C09142=1180.504,309.494,-71.507,-176.660,7.868,148.547
C09143=1180.508,309.245,-71.477,-176.662,7.865,148.546
C09144=1180.512,308.997,-71.446,-176.664,7.862,148.546
C09145=1180.517,308.749,-71.415,-176.667,7.859,148.546
C09146=1180.521,308.501,-71.384,-176.669,7.855,148.546
C09147=1180.525,308.253,-71.354,-176.672,7.853,148.546
C09148=1180.529,308.005,-71.323,-176.674,7.850,148.546
C09149=1180.534,307.757,-71.292,-176.677,7.847,148.546
C09150=1180.537,307.509,-71.262,-176.679,7.844,148.546
C09151=1180.542,307.261,-71.231,-176.682,7.841,148.546
C09152=1180.546,307.013,-71.200,-176.685,7.838,148.546
C09153=1180.550,306.765,-71.170,-176.687,7.835,148.546
C09154=1180.555,306.516,-71.140,-176.690,7.832,148.546
C09155=1180.559,306.268,-71.109,-176.692,7.829,148.546
C09156=1180.563,306.020,-71.079,-176.695,7.826,148.546
C09157=1180.568,305.772,-71.048,-176.697,7.823,148.546
C09158=1180.572,305.525,-71.018,-176.700,7.820,148.546
C09159=1180.576,305.276,-70.987,-176.702,7.817,148.546
C09160=1180.580,305.027,-70.956,-176.705,7.814,148.546
C09161=1180.584,304.780,-70.926,-176.707,7.811,148.546
C09162=1180.589,304.532,-70.896,-176.710,7.808,148.546
C09163=1180.593,304.284,-70.865,-176.713,7.805,148.546
C09164=1180.597,304.035,-70.835,-176.716,7.802,148.546
C09165=1180.601,303.787,-70.805,-176.717,7.799,148.546
C09166=1180.606,303.539,-70.774,-176.720,7.796,148.546
C09167=1180.610,303.292,-70.744,-176.723,7.793,148.546
C09168=1180.614,303.043,-70.714,-176.725,7.790,148.546
C09169=1180.618,302.795,-70.684,-176.728,7.787,148.546
C09170=1180.622,302.547,-70.653,-176.730,7.784,148.546
C09171=1180.627,302.299,-70.623,-176.733,7.781,148.546
C09172=1180.631,302.051,-70.592,-176.736,7.778,148.546
C09173=1180.635,301.802,-70.563,-176.738,7.776,148.545
C09174=1180.640,301.554,-70.532,-176.740,7.773,148.545
C09175=1180.644,301.307,-70.502,-176.743,7.770,148.545
C09176=1180.649,301.058,-70.472,-176.746,7.767,148.545
C09177=1180.652,300.810,-70.441,-176.748,7.764,148.546
C09178=1180.657,300.561,-70.411,-176.751,7.760,148.545
C09179=1180.661,300.314,-70.381,-176.753,7.757,148.545
C09180=1180.666,300.065,-70.351,-176.756,7.755,148.545
C09181=1180.670,299.817,-70.321,-176.758,7.752,148.545
C09182=1180.674,299.569,-70.291,-176.761,7.749,148.545
C09183=1180.678,299.321,-70.261,-176.763,7.746,148.545
C09184=1180.683,299.073,-70.231,-176.766,7.743,148.545
C09185=1180.686,298.825,-70.201,-176.769,7.740,148.545
C09186=1180.691,298.576,-70.171,-176.771,7.737,148.545
C09187=1180.695,298.328,-70.140,-176.774,7.735,148.545
C09188=1180.700,298.080,-70.110,-176.776,7.731,148.545
C09189=1180.703,297.832,-70.080,-176.779,7.728,148.545
C09190=1180.708,297.584,-70.051,-176.781,7.726,148.545
C09191=1180.713,297.335,-70.021,-176.784,7.723,148.545
C09192=1180.716,297.088,-69.991,-176.787,7.720,148.545
C09193=1180.721,296.839,-69.961,-176.789,7.717,148.545
C09194=1180.725,296.591,-69.932,-176.791,7.714,148.545
C09195=1180.729,296.343,-69.901,-176.794,7.711,148.545
C09196=1180.734,296.095,-69.871,-176.797,7.708,148.545
C09197=1180.738,295.846,-69.842,-176.799,7.705,148.545
C09198=1180.742,295.599,-69.812,-176.802,7.702,148.545
C09199=1180.747,295.350,-69.782,-176.805,7.699,148.545
C09200=1180.751,295.102,-69.752,-176.807,7.697,148.545
C09201=1180.755,294.854,-69.722,-176.809,7.694,148.545
C09202=1180.759,294.606,-69.693,-176.812,7.691,148.545
C09203=1180.764,294.358,-69.663,-176.815,7.688,148.545
C09204=1180.768,294.109,-69.633,-176.817,7.685,148.545
C09205=1180.772,293.861,-69.604,-176.820,7.682,148.545
C09206=1180.776,293.613,-69.574,-176.822,7.680,148.545
C09207=1180.780,293.365,-69.544,-176.825,7.677,148.545
C09208=1180.785,293.116,-69.514,-176.827,7.673,148.545
C09209=1180.789,292.868,-69.485,-176.830,7.670,148.545
C09210=1180.793,292.620,-69.455,-176.833,7.667,148.545
C09211=1180.798,292.372,-69.426,-176.835,7.665,148.545
C09212=1180.801,292.124,-69.396,-176.838,7.662,148.545
C09213=1180.806,291.876,-69.366,-176.840,7.659,148.545
C09214=1180.810,291.627,-69.337,-176.843,7.656,148.545
C09215=1180.815,291.379,-69.307,-176.846,7.653,148.545
C09216=1180.819,291.131,-69.277,-176.848,7.650,148.545
C09217=1180.823,290.882,-69.248,-176.850,7.648,148.545
C09218=1180.827,290.634,-69.218,-176.853,7.645,148.545
C09219=1180.832,290.387,-69.189,-176.856,7.642,148.545
C09220=1180.836,290.138,-69.160,-176.858,7.639,148.545
C09221=1180.840,289.890,-69.130,-176.861,7.636,148.546
C09222=1180.845,289.642,-69.101,-176.863,7.634,148.546
C09223=1180.849,289.393,-69.071,-176.866,7.631,148.546
C09224=1180.853,289.145,-69.042,-176.869,7.628,148.546
C09225=1180.857,288.897,-69.012,-176.871,7.625,148.546
C09226=1180.863,288.622,-68.980,-176.874,7.622,148.546
C09227=1180.867,288.348,-68.947,-176.877,7.619,148.546
C09228=1180.872,288.072,-68.915,-176.880,7.616,148.546
C09229=1180.876,287.799,-68.883,-176.883,7.612,148.546
C09230=1180.881,287.550,-68.854,-176.885,7.610,148.546
C09231=1180.885,287.302,-68.824,-176.888,7.607,148.546
C09232=1180.889,287.053,-68.795,-176.890,7.603,148.546
C09233=1180.894,286.806,-68.766,-176.893,7.600,148.546
C09234=1180.898,286.557,-68.736,-176.896,7.597,148.546
C09235=1180.902,286.309,-68.707,-176.898,7.595,148.546
C09236=1180.907,286.060,-68.678,-176.900,7.592,148.546
C09237=1180.911,285.812,-68.649,-176.903,7.589,148.546
C09238=1180.915,285.564,-68.619,-176.906,7.586,148.546
C09239=1180.920,285.316,-68.590,-176.909,7.583,148.546
C09240=1180.924,285.067,-68.561,-176.911,7.581,148.546
C09241=1180.928,284.819,-68.532,-176.913,7.578,148.546
C09242=1180.933,284.571,-68.503,-176.916,7.575,148.546
C09243=1180.937,284.322,-68.473,-176.919,7.572,148.546
C09244=1180.941,284.075,-68.445,-176.921,7.570,148.546
C09245=1180.945,283.826,-68.416,-176.924,7.567,148.546
C09246=1180.949,283.578,-68.386,-176.927,7.564,148.546
C09247=1180.954,283.329,-68.358,-176.929,7.561,148.546
C09248=1180.959,283.082,-68.329,-176.932,7.558,148.546
C09249=1180.963,282.833,-68.299,-176.934,7.556,148.546
C09250=1180.967,282.584,-68.270,-176.937,7.553,148.546
C09251=1180.971,282.337,-68.241,-176.940,7.550,148.546
C09252=1180.976,282.088,-68.213,-176.942,7.547,148.547
C09253=1180.980,281.840,-68.184,-176.945,7.545,148.547
C09254=1180.984,281.592,-68.154,-176.947,7.542,148.547
C09255=1180.989,281.343,-68.125,-176.950,7.539,148.547
C09256=1180.993,281.096,-68.097,-176.953,7.536,148.547
C09257=1180.997,280.847,-68.068,-176.955,7.534,148.547
C09258=1181.001,280.598,-68.039,-176.958,7.531,148.547
C09259=1181.006,280.350,-68.010,-176.960,7.528,148.547
C09260=1181.010,280.102,-67.982,-176.963,7.525,148.547
C09261=1181.014,279.853,-67.953,-176.965,7.522,148.547
C09262=1181.019,279.605,-67.923,-176.968,7.520,148.547
C09263=1181.024,279.357,-67.895,-176.971,7.517,148.547
C09264=1181.027,279.109,-67.866,-176.973,7.514,148.547
C09265=1181.032,278.860,-67.837,-176.976,7.511,148.547
C09266=1181.037,278.612,-67.809,-176.978,7.508,148.547
C09267=1181.040,278.364,-67.780,-176.981,7.505,148.547
C09268=1181.045,278.115,-67.751,-176.984,7.502,148.547
C09269=1181.049,277.868,-67.722,-176.986,7.500,148.547
C09270=1181.053,277.619,-67.694,-176.989,7.497,148.547
C09271=1181.058,277.370,-67.665,-176.991,7.494,148.547
C09272=1181.063,277.123,-67.636,-176.994,7.491,148.548
C09273=1181.066,276.874,-67.608,-176.996,7.489,148.548
C09274=1181.071,276.625,-67.579,-176.999,7.486,148.548
C09275=1181.075,276.377,-67.552,-177.002,7.483,148.548
C09276=1181.079,276.129,-67.522,-177.004,7.481,148.548
C09277=1181.084,275.880,-67.494,-177.007,7.478,148.548
C09278=1181.088,275.632,-67.466,-177.009,7.475,148.548
C09279=1181.092,275.384,-67.436,-177.012,7.472,148.548
C09280=1181.097,275.136,-67.409,-177.014,7.470,148.548
C09281=1181.101,274.887,-67.380,-177.017,7.467,148.548
C09282=1181.105,274.639,-67.352,-177.020,7.464,148.548
C09283=1181.110,274.390,-67.323,-177.022,7.462,148.548
C09284=1181.114,274.142,-67.294,-177.025,7.459,148.548
C09285=1181.119,273.894,-67.266,-177.027,7.456,148.548
C09286=1181.123,273.645,-67.237,-177.030,7.453,148.548
C09287=1181.127,273.397,-67.210,-177.032,7.451,148.548
C09288=1181.132,273.149,-67.181,-177.035,7.448,148.549
C09289=1181.136,272.900,-67.153,-177.038,7.445,148.549
C09290=1181.141,272.652,-67.124,-177.040,7.443,148.549
C09291=1181.144,272.404,-67.095,-177.043,7.440,148.549
C09292=1181.149,272.156,-67.067,-177.046,7.437,148.549
C09293=1181.153,271.907,-67.039,-177.049,7.434,148.549
C09294=1181.157,271.659,-67.011,-177.051,7.432,148.549
C09295=1181.162,271.410,-66.982,-177.053,7.429,148.549
C09296=1181.166,271.162,-66.955,-177.056,7.426,148.549
C09297=1181.171,270.914,-66.926,-177.058,7.424,148.549
C09298=1181.175,270.666,-66.898,-177.061,7.421,148.549
C09299=1181.179,270.417,-66.869,-177.064,7.418,148.549
C09300=1181.184,270.169,-66.842,-177.066,7.416,148.549
C09301=1181.188,269.920,-66.813,-177.069,7.413,148.550
C09302=1181.193,269.672,-66.785,-177.072,7.410,148.550
C09303=1181.196,269.424,-66.757,-177.074,7.408,148.550
C09304=1181.201,269.175,-66.729,-177.077,7.405,148.550
C09305=1181.205,268.927,-66.700,-177.080,7.402,148.550
C09306=1181.210,268.678,-66.673,-177.082,7.399,148.550
C09307=1181.214,268.429,-66.645,-177.084,7.397,148.550
C09308=1181.219,268.182,-66.617,-177.087,7.394,148.550
C09309=1181.222,267.933,-66.589,-177.090,7.391,148.550
C09310=1181.228,267.685,-66.560,-177.093,7.389,148.550
C09311=1181.231,267.436,-66.532,-177.095,7.386,148.550
C09312=1181.236,267.188,-66.504,-177.098,7.383,148.550
C09313=1181.241,266.940,-66.477,-177.100,7.381,148.550
C09314=1181.245,266.691,-66.449,-177.103,7.378,148.551
C09315=1181.249,266.443,-66.421,-177.106,7.375,148.551
C09316=1181.254,266.194,-66.392,-177.108,7.373,148.551
C09317=1181.258,265.946,-66.365,-177.111,7.370,148.551
C09318=1181.262,265.697,-66.337,-177.114,7.367,148.551
C09319=1181.266,265.449,-66.309,-177.116,7.365,148.551
C09320=1181.271,265.201,-66.281,-177.119,7.362,148.551
C09321=1181.276,264.952,-66.253,-177.121,7.359,148.551
C09322=1181.280,264.704,-66.226,-177.124,7.357,148.551
C09323=1181.284,264.456,-66.198,-177.126,7.354,148.551
C09324=1181.289,264.207,-66.170,-177.129,7.352,148.552
C09325=1181.293,263.959,-66.142,-177.132,7.349,148.552
C09326=1181.297,263.710,-66.114,-177.134,7.346,148.552
C09327=1181.302,263.462,-66.087,-177.137,7.344,148.552
C09328=1181.306,263.214,-66.059,-177.139,7.341,148.552
C09329=1181.310,262.965,-66.031,-177.142,7.338,148.552
C09330=1181.315,262.693,-66.001,-177.145,7.335,148.552
C09331=1181.320,262.419,-65.970,-177.148,7.332,148.552
C09332=1181.325,262.147,-65.940,-177.151,7.329,148.552
C09333=1181.330,261.873,-65.909,-177.154,7.327,148.553
C09334=1181.334,261.625,-65.882,-177.156,7.324,148.553
C09335=1181.338,261.376,-65.854,-177.159,7.321,148.553
C09336=1181.343,261.128,-65.827,-177.161,7.318,148.553
C09337=1181.347,260.880,-65.799,-177.164,7.316,148.553
C09338=1181.351,260.631,-65.771,-177.167,7.314,148.553
C09339=1181.356,260.383,-65.744,-177.169,7.311,148.553
C09340=1181.361,260.134,-65.716,-177.172,7.308,148.553
C09341=1181.365,259.886,-65.688,-177.174,7.306,148.553
C09342=1181.369,259.637,-65.661,-177.177,7.303,148.553
C09343=1181.374,259.389,-65.633,-177.180,7.301,148.554
C09344=1181.378,259.141,-65.606,-177.183,7.298,148.554
C09345=1181.382,258.891,-65.578,-177.185,7.296,148.554
C09346=1181.387,258.643,-65.551,-177.188,7.293,148.554
C09347=1181.391,258.395,-65.524,-177.190,7.290,148.554
C09348=1181.396,258.147,-65.496,-177.193,7.288,148.554
C09349=1181.400,257.898,-65.468,-177.196,7.285,148.554
C09350=1181.405,257.649,-65.441,-177.198,7.283,148.554
C09351=1181.409,257.402,-65.414,-177.201,7.280,148.554
C09352=1181.414,257.153,-65.387,-177.203,7.278,148.555
C09353=1181.418,256.904,-65.359,-177.206,7.275,148.555
C09354=1181.422,256.655,-65.332,-177.209,7.272,148.555
C09355=1181.427,256.407,-65.304,-177.211,7.270,148.555
C09356=1181.431,256.159,-65.277,-177.214,7.267,148.555
C09357=1181.435,255.910,-65.250,-177.216,7.265,148.555
C09358=1181.440,255.662,-65.222,-177.219,7.262,148.555
C09359=1181.444,255.414,-65.196,-177.222,7.259,148.555
C09360=1181.448,255.165,-65.168,-177.224,7.257,148.555
C09361=1181.453,254.917,-65.141,-177.227,7.254,148.556
C09362=1181.457,254.668,-65.114,-177.229,7.252,148.556
C09363=1181.461,254.420,-65.086,-177.232,7.249,148.556
C09364=1181.466,254.171,-65.059,-177.235,7.246,148.556
C09365=1181.471,253.923,-65.032,-177.237,7.244,148.556
C09366=1181.475,253.674,-65.005,-177.240,7.241,148.556
C09367=1181.480,253.426,-64.978,-177.242,7.239,148.556
C09368=1181.483,253.177,-64.951,-177.245,7.236,148.557
C09369=1181.488,252.928,-64.924,-177.248,7.234,148.557
C09370=1181.492,252.680,-64.896,-177.250,7.231,148.557
C09371=1181.497,252.432,-64.869,-177.253,7.228,148.557
C09372=1181.502,252.183,-64.842,-177.256,7.227,148.557
C09373=1181.506,251.935,-64.815,-177.258,7.224,148.557
C09374=1181.510,251.687,-64.789,-177.261,7.221,148.557
C09375=1181.514,251.438,-64.761,-177.263,7.218,148.557
C09376=1181.519,251.189,-64.734,-177.266,7.217,148.558
C09377=1181.524,250.941,-64.707,-177.269,7.214,148.558
C09378=1181.527,250.692,-64.681,-177.271,7.211,148.558
C09379=1181.532,250.444,-64.654,-177.274,7.209,148.558
C09380=1181.537,250.195,-64.626,-177.277,7.206,148.558
C09381=1181.541,249.947,-64.599,-177.279,7.204,148.558
C09382=1181.545,249.699,-64.573,-177.282,7.201,148.559
C09383=1181.550,249.450,-64.546,-177.284,7.199,148.559
C09384=1181.555,249.202,-64.519,-177.287,7.196,148.559
C09385=1181.559,248.952,-64.492,-177.290,7.194,148.559
C09386=1181.563,248.704,-64.466,-177.293,7.191,148.559
C09387=1181.568,248.455,-64.439,-177.295,7.189,148.559
C09388=1181.572,248.207,-64.412,-177.297,7.186,148.559
C09389=1181.576,247.959,-64.385,-177.300,7.184,148.560
C09390=1181.581,247.710,-64.358,-177.303,7.181,148.560
C09391=1181.585,247.462,-64.331,-177.306,7.178,148.560
C09392=1181.590,247.213,-64.305,-177.308,7.176,148.560
C09393=1181.594,246.964,-64.278,-177.311,7.173,148.560
C09394=1181.599,246.716,-64.251,-177.313,7.171,148.560
C09395=1181.603,246.468,-64.225,-177.316,7.169,148.560
C09396=1181.608,246.219,-64.198,-177.318,7.167,148.561
C09397=1181.612,245.970,-64.172,-177.322,7.164,148.561
C09398=1181.616,245.722,-64.145,-177.324,7.162,148.561
C09399=1181.621,245.473,-64.118,-177.327,7.159,148.561
C09400=1181.625,245.225,-64.091,-177.329,7.157,148.561
C09401=1181.630,244.976,-64.065,-177.332,7.154,148.561
C09402=1181.634,244.728,-64.038,-177.334,7.152,148.561
C09403=1181.639,244.479,-64.011,-177.337,7.149,148.562
C09404=1181.644,244.230,-63.985,-177.340,7.147,148.562
C09405=1181.647,243.982,-63.959,-177.342,7.144,148.562
C09406=1181.652,243.734,-63.931,-177.345,7.142,148.562
C09407=1181.656,243.485,-63.906,-177.348,7.139,148.562
C09408=1181.661,243.236,-63.879,-177.350,7.137,148.563
C09409=1181.665,242.988,-63.852,-177.353,7.134,148.563
C09410=1181.670,242.739,-63.826,-177.355,7.132,148.563
C09411=1181.674,242.491,-63.799,-177.358,7.130,148.563
C09412=1181.679,242.242,-63.773,-177.361,7.128,148.563
C09413=1181.683,241.993,-63.747,-177.363,7.125,148.563
C09414=1181.688,241.744,-63.720,-177.366,7.123,148.564
C09415=1181.692,241.496,-63.694,-177.369,7.120,148.564
C09416=1181.697,241.248,-63.667,-177.371,7.118,148.564
C09417=1181.701,241.000,-63.641,-177.374,7.115,148.564
C09418=1181.705,240.751,-63.615,-177.376,7.113,148.564
C09419=1181.710,240.502,-63.588,-177.379,7.110,148.564
C09420=1181.714,240.254,-63.562,-177.382,7.108,148.565
C09421=1181.719,240.005,-63.536,-177.385,7.105,148.565
C09422=1181.723,239.756,-63.510,-177.387,7.103,148.565
C09423=1181.728,239.508,-63.483,-177.390,7.100,148.565
C09424=1181.732,239.259,-63.457,-177.392,7.098,148.565
C09425=1181.736,239.011,-63.431,-177.395,7.095,148.565
C09426=1181.741,238.762,-63.405,-177.398,7.094,148.566
C09427=1181.745,238.514,-63.378,-177.401,7.091,148.566
C09428=1181.750,238.265,-63.352,-177.403,7.089,148.566
C09429=1181.754,238.016,-63.326,-177.405,7.087,148.566
C09430=1181.758,237.768,-63.300,-177.408,7.084,148.566
C09431=1181.763,237.519,-63.273,-177.411,7.082,148.567
C09432=1181.768,237.270,-63.248,-177.414,7.079,148.567
C09433=1181.772,237.023,-63.221,-177.416,7.077,148.567
C09434=1181.778,236.750,-63.193,-177.419,7.074,148.567
C09435=1181.782,236.479,-63.164,-177.422,7.072,148.567
C09436=1181.787,236.207,-63.136,-177.425,7.069,148.567
C09437=1181.791,235.936,-63.107,-177.428,7.067,148.568
C09438=1181.797,235.687,-63.081,-177.431,7.064,148.568
C09439=1181.801,235.439,-63.056,-177.433,7.062,148.568
C09440=1181.805,235.190,-63.030,-177.436,7.059,148.568
C09441=1181.809,234.942,-63.003,-177.438,7.057,148.568
C09442=1181.814,234.693,-62.977,-177.441,7.054,148.569
C09443=1181.819,234.444,-62.952,-177.444,7.052,148.569
C09444=1181.823,234.196,-62.926,-177.446,7.050,148.569
C09445=1181.827,233.947,-62.900,-177.449,7.048,148.569
C09446=1181.832,233.698,-62.874,-177.451,7.045,148.569
C09447=1181.836,233.450,-62.847,-177.454,7.043,148.570
C09448=1181.841,233.201,-62.822,-177.457,7.041,148.570
C09449=1181.845,232.953,-62.796,-177.460,7.038,148.570
C09450=1181.849,232.704,-62.770,-177.462,7.036,148.570
C09451=1181.854,232.455,-62.744,-177.465,7.033,148.570
C09452=1181.859,232.207,-62.719,-177.467,7.031,148.571
C09453=1181.863,231.958,-62.693,-177.470,7.029,148.571
C09454=1181.868,231.709,-62.667,-177.473,7.026,148.571
C09455=1181.872,231.461,-62.642,-177.475,7.025,148.571
C09456=1181.877,231.212,-62.616,-177.478,7.022,148.571
C09457=1181.881,230.963,-62.590,-177.481,7.020,148.572
C09458=1181.886,230.714,-62.564,-177.483,7.018,148.572
C09459=1181.891,230.466,-62.539,-177.486,7.015,148.572
C09460=1181.895,230.217,-62.513,-177.488,7.013,148.572
C09461=1181.899,229.968,-62.487,-177.492,7.010,148.573
C09462=1181.904,229.720,-62.462,-177.494,7.008,148.573
C09463=1181.908,229.472,-62.436,-177.496,7.006,148.573
C09464=1181.912,229.223,-62.410,-177.499,7.003,148.573
C09465=1181.917,228.974,-62.384,-177.502,7.001,148.573
C09466=1181.921,228.726,-62.359,-177.505,6.999,148.573
C09467=1181.926,228.477,-62.333,-177.507,6.997,148.574
C09468=1181.930,228.228,-62.308,-177.509,6.995,148.574
C09469=1181.935,227.980,-62.282,-177.513,6.992,148.574
C09470=1181.939,227.731,-62.256,-177.515,6.990,148.574
C09471=1181.944,227.483,-62.232,-177.518,6.987,148.575
C09472=1181.948,227.234,-62.206,-177.521,6.985,148.575
C09473=1181.952,226.985,-62.180,-177.523,6.983,148.575
C09474=1181.957,226.737,-62.155,-177.526,6.981,148.575
C09475=1181.962,226.488,-62.129,-177.528,6.978,148.575
C09476=1181.966,226.239,-62.103,-177.532,6.976,148.576
C09477=1181.971,225.991,-62.079,-177.534,6.974,148.576
C09478=1181.975,225.742,-62.053,-177.536,6.972,148.576
C09479=1181.979,225.493,-62.027,-177.539,6.969,148.576
C09480=1181.984,225.245,-62.002,-177.542,6.967,148.577
C09481=1181.989,224.995,-61.977,-177.544,6.965,148.577
C09482=1181.994,224.747,-61.951,-177.547,6.962,148.577
C09483=1181.998,224.498,-61.926,-177.550,6.960,148.577
C09484=1182.003,224.250,-61.900,-177.553,6.958,148.577
C09485=1182.007,224.001,-61.875,-177.555,6.956,148.578
C09486=1182.011,223.752,-61.849,-177.557,6.954,148.578
C09487=1182.016,223.504,-61.824,-177.561,6.951,148.578
C09488=1182.021,223.255,-61.799,-177.563,6.949,148.578
C09489=1182.025,223.007,-61.774,-177.565,6.947,148.579
C09490=1182.029,222.757,-61.749,-177.569,6.944,148.579
C09491=1182.034,222.509,-61.724,-177.571,6.942,148.579
C09492=1182.038,222.260,-61.698,-177.574,6.940,148.579
C09493=1182.043,222.011,-61.673,-177.576,6.937,148.579
C09494=1182.048,221.763,-61.648,-177.579,6.936,148.580
C09495=1182.052,221.514,-61.623,-177.582,6.933,148.580
C09496=1182.056,221.266,-61.598,-177.584,6.931,148.580
C09497=1182.061,221.017,-61.572,-177.587,6.929,148.580
C09498=1182.066,220.768,-61.547,-177.590,6.926,148.581
C09499=1182.070,220.519,-61.522,-177.592,6.924,148.581
C09500=1182.074,220.271,-61.498,-177.595,6.922,148.581
C09501=1182.079,220.022,-61.472,-177.598,6.919,148.581
C09502=1182.084,219.773,-61.447,-177.600,6.918,148.582
C09503=1182.088,219.525,-61.421,-177.603,6.916,148.582
C09504=1182.093,219.276,-61.397,-177.606,6.913,148.582
C09505=1182.097,219.027,-61.372,-177.608,6.911,148.582
C09506=1182.102,218.779,-61.347,-177.611,6.909,148.582
C09507=1182.106,218.529,-61.322,-177.614,6.906,148.583
C09508=1182.110,218.282,-61.297,-177.617,6.905,148.583
C09509=1182.115,218.032,-61.272,-177.619,6.902,148.583
C09510=1182.120,217.784,-61.247,-177.622,6.900,148.584
C09511=1182.124,217.535,-61.222,-177.625,6.898,148.584
C09512=1182.129,217.286,-61.198,-177.627,6.896,148.584
C09513=1182.133,217.038,-61.172,-177.630,6.893,148.584
C09514=1182.138,216.789,-61.147,-177.632,6.891,148.584
C09515=1182.142,216.540,-61.123,-177.635,6.889,148.585
C09516=1182.147,216.291,-61.097,-177.638,6.887,148.585
C09517=1182.152,216.043,-61.073,-177.640,6.884,148.585
C09518=1182.155,215.794,-61.048,-177.643,6.883,148.586
C09519=1182.160,215.545,-61.023,-177.646,6.880,148.586
C09520=1182.165,215.297,-60.998,-177.648,6.878,148.586
C09521=1182.169,215.048,-60.974,-177.651,6.876,148.586
C09522=1182.174,214.799,-60.949,-177.654,6.874,148.587
C09523=1182.178,214.550,-60.924,-177.656,6.871,148.587
C09524=1182.183,214.302,-60.899,-177.659,6.870,148.587
C09525=1182.188,214.053,-60.875,-177.662,6.868,148.587
C09526=1182.192,213.804,-60.850,-177.664,6.865,148.587
C09527=1182.197,213.555,-60.825,-177.667,6.863,148.588
C09528=1182.200,213.307,-60.800,-177.670,6.861,148.588
C09529=1182.206,213.058,-60.776,-177.673,6.858,148.588
C09530=1182.210,212.809,-60.751,-177.675,6.856,148.589
C09531=1182.215,212.560,-60.726,-177.678,6.855,148.589
C09532=1182.219,212.312,-60.702,-177.680,6.852,148.589
C09533=1182.224,212.063,-60.678,-177.683,6.850,148.589
C09534=1182.229,211.813,-60.653,-177.686,6.848,148.590
C09535=1182.233,211.566,-60.628,-177.688,6.846,148.590
C09536=1182.238,211.317,-60.603,-177.691,6.843,148.590
C09537=1182.242,211.068,-60.579,-177.694,6.841,148.590
C09538=1182.247,210.798,-60.552,-177.697,6.840,148.591
C09539=1182.252,210.527,-60.526,-177.699,6.837,148.591
C09540=1182.257,210.256,-60.499,-177.703,6.834,148.591
C09541=1182.262,209.986,-60.472,-177.705,6.832,148.592
C09542=1182.266,209.737,-60.448,-177.708,6.831,148.592
C09543=1182.271,209.489,-60.424,-177.711,6.828,148.592
C09544=1182.275,209.240,-60.399,-177.713,6.826,148.592
C09545=1182.280,208.991,-60.375,-177.716,6.824,148.593
C09546=1182.285,208.742,-60.350,-177.719,6.822,148.593
C09547=1182.289,208.493,-60.326,-177.721,6.819,148.593
C09548=1182.294,208.245,-60.301,-177.724,6.817,148.593
C09549=1182.298,207.996,-60.277,-177.727,6.816,148.594
C09550=1182.302,207.748,-60.253,-177.729,6.813,148.594
C09551=1182.307,207.498,-60.228,-177.732,6.811,148.594
C09552=1182.312,207.249,-60.205,-177.735,6.809,148.595
C09553=1182.317,207.001,-60.180,-177.737,6.807,148.595
C09554=1182.321,206.752,-60.156,-177.740,6.804,148.595
C09555=1182.325,206.503,-60.132,-177.743,6.802,148.595
C09556=1182.330,206.254,-60.107,-177.746,6.801,148.596
C09557=1182.335,206.006,-60.083,-177.748,6.799,148.596
C09558=1182.339,205.758,-60.059,-177.751,6.796,148.596
C09559=1182.344,205.508,-60.035,-177.754,6.794,148.596
C09560=1182.348,205.259,-60.010,-177.756,6.792,148.597
C09561=1182.353,205.011,-59.986,-177.758,6.790,148.597
C09562=1182.358,204.762,-59.962,-177.762,6.788,148.597
C09563=1182.362,204.513,-59.938,-177.764,6.786,148.598
C09564=1182.367,204.265,-59.914,-177.767,6.784,148.598
C09565=1182.371,204.015,-59.890,-177.769,6.782,148.598
C09566=1182.376,203.767,-59.865,-177.772,6.780,148.598
C09567=1182.380,203.518,-59.842,-177.775,6.777,148.599
C09568=1182.385,203.269,-59.818,-177.778,6.776,148.599
C09569=1182.389,203.021,-59.794,-177.780,6.774,148.599
C09570=1182.394,202.771,-59.768,-177.783,6.772,148.599
C09571=1182.398,202.522,-59.745,-177.786,6.769,148.600
C09572=1182.403,202.274,-59.721,-177.788,6.767,148.600
C09573=1182.407,202.026,-59.697,-177.791,6.765,148.600
C09574=1182.413,201.776,-59.673,-177.793,6.763,148.601
C09575=1182.417,201.528,-59.649,-177.796,6.762,148.601
C09576=1182.422,201.279,-59.626,-177.799,6.759,148.601
C09577=1182.426,201.030,-59.601,-177.801,6.757,148.601
C09578=1182.430,200.781,-59.577,-177.804,6.755,148.602
C09579=1182.435,200.532,-59.554,-177.807,6.753,148.602
C09580=1182.440,200.283,-59.529,-177.810,6.751,148.602
C09581=1182.444,200.034,-59.506,-177.812,6.748,148.603
C09582=1182.449,199.786,-59.482,-177.815,6.747,148.603
C09583=1182.454,199.537,-59.458,-177.818,6.745,148.603
C09584=1182.458,199.289,-59.434,-177.820,6.743,148.604
C09585=1182.463,199.040,-59.411,-177.823,6.740,148.604
C09586=1182.466,198.790,-59.386,-177.826,6.738,148.604
C09587=1182.472,198.541,-59.362,-177.828,6.737,148.604
C09588=1182.476,198.293,-59.338,-177.831,6.735,148.605
C09589=1182.481,198.044,-59.315,-177.834,6.733,148.605
C09590=1182.485,197.795,-59.291,-177.836,6.731,148.605
C09591=1182.490,197.546,-59.268,-177.839,6.728,148.606
C09592=1182.494,197.298,-59.243,-177.842,6.726,148.606
C09593=1182.499,197.049,-59.220,-177.844,6.725,148.606
C09594=1182.504,196.800,-59.197,-177.847,6.723,148.607
C09595=1182.508,196.551,-59.173,-177.849,6.721,148.607
C09596=1182.513,196.302,-59.149,-177.852,6.718,148.607
C09597=1182.517,196.054,-59.125,-177.855,6.716,148.607
C09598=1182.522,195.805,-59.102,-177.858,6.715,148.608
C09599=1182.527,195.556,-59.079,-177.860,6.712,148.608
C09600=1182.531,195.307,-59.054,-177.863,6.711,148.608
C09601=1182.536,195.058,-59.031,-177.865,6.709,148.609
C09602=1182.541,194.809,-59.008,-177.869,6.706,148.609
C09603=1182.545,194.561,-58.984,-177.871,6.704,148.609
C09604=1182.550,194.312,-58.960,-177.874,6.703,148.610
C09605=1182.554,194.063,-58.937,-177.876,6.700,148.610
C09606=1182.559,193.814,-58.914,-177.879,6.699,148.610
C09607=1182.563,193.565,-58.890,-177.881,6.697,148.610
C09608=1182.568,193.316,-58.866,-177.885,6.694,148.611
C09609=1182.573,193.067,-58.843,-177.887,6.692,148.611
C09610=1182.578,192.818,-58.819,-177.889,6.690,148.611
C09611=1182.582,192.570,-58.795,-177.892,6.689,148.612
C09612=1182.587,192.321,-58.772,-177.895,6.687,148.612
C09613=1182.591,192.072,-58.749,-177.897,6.685,148.612
C09614=1182.596,191.823,-58.725,-177.901,6.682,148.613
C09615=1182.600,191.574,-58.703,-177.903,6.681,148.613
C09616=1182.605,191.325,-58.679,-177.906,6.678,148.613
C09617=1182.609,191.077,-58.655,-177.908,6.677,148.613
C09618=1182.614,190.828,-58.632,-177.911,6.675,148.614
C09619=1182.619,190.579,-58.608,-177.914,6.673,148.614
C09620=1182.623,190.330,-58.585,-177.916,6.671,148.614
C09621=1182.628,190.080,-58.562,-177.919,6.669,148.615
C09622=1182.632,189.832,-58.539,-177.922,6.667,148.615
C09623=1182.637,189.583,-58.516,-177.924,6.665,148.615
C09624=1182.642,189.334,-58.493,-177.927,6.663,148.616
C09625=1182.647,189.085,-58.469,-177.930,6.661,148.616
C09626=1182.651,188.836,-58.446,-177.932,6.659,148.616
C09627=1182.656,188.587,-58.422,-177.935,6.658,148.617
C09628=1182.660,188.339,-58.400,-177.938,6.656,148.617
C09629=1182.665,188.090,-58.376,-177.940,6.653,148.617
C09630=1182.669,187.841,-58.353,-177.943,6.651,148.617
C09631=1182.675,187.592,-58.330,-177.946,6.649,148.618
C09632=1182.679,187.343,-58.307,-177.948,6.648,148.618
C09633=1182.683,187.094,-58.284,-177.951,6.646,148.619
C09634=1182.688,186.845,-58.261,-177.954,6.644,148.619
C09635=1182.693,186.596,-58.237,-177.956,6.642,148.619
C09636=1182.697,186.348,-58.214,-177.959,6.640,148.619
C09637=1182.701,186.099,-58.191,-177.961,6.638,148.620
C09638=1182.707,185.850,-58.168,-177.965,6.636,148.620
C09639=1182.711,185.601,-58.145,-177.967,6.634,148.620
C09640=1182.715,185.353,-58.122,-177.970,6.632,148.621
C09641=1182.720,185.104,-58.099,-177.973,6.630,148.621
C09642=1182.725,184.834,-58.074,-177.975,6.628,148.622
C09643=1182.730,184.564,-58.049,-177.979,6.626,148.622
C09644=1182.735,184.295,-58.024,-177.981,6.624,148.622
C09645=1182.740,184.025,-58.000,-177.984,6.622,148.623
C09646=1182.745,183.776,-57.976,-177.987,6.621,148.623
C09647=1182.749,183.527,-57.953,-177.989,6.619,148.623
C09648=1182.754,183.278,-57.931,-177.992,6.616,148.624
C09649=1182.759,183.029,-57.908,-177.995,6.614,148.624
C09650=1182.763,182.780,-57.884,-177.997,6.612,148.624
C09651=1182.767,182.532,-57.862,-178.000,6.610,148.624
C09652=1182.772,182.282,-57.839,-178.003,6.609,148.625
C09653=1182.777,182.034,-57.817,-178.005,6.607,148.625
C09654=1182.782,181.785,-57.793,-178.008,6.605,148.626
C09655=1182.787,181.535,-57.771,-178.011,6.603,148.626
C09656=1182.791,181.287,-57.748,-178.013,6.602,148.626
C09657=1182.796,181.038,-57.725,-178.016,6.600,148.627
C09658=1182.800,180.789,-57.702,-178.019,6.598,148.627
C09659=1182.805,180.540,-57.680,-178.021,6.596,148.627
C09660=1182.809,180.291,-57.657,-178.024,6.593,148.627
C09661=1182.814,180.043,-57.634,-178.027,6.591,148.628
C09662=1182.818,179.793,-57.612,-178.029,6.590,148.628
C09663=1182.823,179.544,-57.588,-178.032,6.588,148.629
C09664=1182.828,179.296,-57.567,-178.035,6.586,148.629
C09665=1182.833,179.047,-57.543,-178.037,6.584,148.629
C09666=1182.837,178.798,-57.521,-178.040,6.583,148.630
C09667=1182.842,178.548,-57.498,-178.043,6.581,148.630
C09668=1182.846,178.300,-57.475,-178.046,6.579,148.630
C09669=1182.851,178.051,-57.453,-178.048,6.577,148.631
C09670=1182.855,177.802,-57.430,-178.051,6.575,148.631
C09671=1182.861,177.553,-57.408,-178.054,6.574,148.631
C09672=1182.865,177.304,-57.385,-178.056,6.572,148.632
C09673=1182.870,177.055,-57.362,-178.059,6.570,148.632
C09674=1182.874,176.807,-57.340,-178.061,6.568,148.632
C09675=1182.879,176.557,-57.317,-178.064,6.566,148.633
C09676=1182.883,176.308,-57.295,-178.066,6.564,148.633
C09677=1182.888,176.060,-57.273,-178.069,6.563,148.633
C09678=1182.893,175.811,-57.250,-178.072,6.561,148.634
C09679=1182.897,175.561,-57.228,-178.074,6.559,148.634
C09680=1182.902,175.313,-57.205,-178.078,6.556,148.634
C09681=1182.907,175.064,-57.182,-178.080,6.555,148.635
C09682=1182.911,174.814,-57.160,-178.083,6.553,148.635
C09683=1182.916,174.566,-57.137,-178.086,6.551,148.635
C09684=1182.921,174.317,-57.115,-178.088,6.549,148.636
C09685=1182.926,174.068,-57.092,-178.091,6.548,148.636
C09686=1182.930,173.819,-57.070,-178.094,6.546,148.637
C09687=1182.934,173.570,-57.048,-178.096,6.544,148.637
C09688=1182.940,173.321,-57.025,-178.099,6.542,148.637
C09689=1182.944,173.072,-57.003,-178.102,6.540,148.638
C09690=1182.949,172.823,-56.982,-178.104,6.539,148.638
C09691=1182.954,172.574,-56.959,-178.107,6.537,148.638
C09692=1182.958,172.325,-56.936,-178.110,6.535,148.639
C09693=1182.963,172.076,-56.914,-178.113,6.533,148.639
C09694=1182.967,171.827,-56.892,-178.115,6.532,148.639
C09695=1182.972,171.579,-56.869,-178.118,6.530,148.640
C09696=1182.977,171.329,-56.847,-178.121,6.528,148.640
C09697=1182.981,171.081,-56.826,-178.123,6.526,148.641
C09698=1182.986,170.831,-56.803,-178.125,6.524,148.641
C09699=1182.991,170.583,-56.781,-178.128,6.522,148.641
C09700=1182.995,170.334,-56.759,-178.131,6.521,148.641
C09701=1183.000,170.084,-56.737,-178.133,6.519,148.642
C09702=1183.005,169.835,-56.714,-178.136,6.517,148.642
C09703=1183.009,169.586,-56.692,-178.139,6.515,148.643
C09704=1183.014,169.337,-56.671,-178.141,6.513,148.643
C09705=1183.018,169.089,-56.648,-178.144,6.512,148.643
C09706=1183.023,168.840,-56.626,-178.147,6.510,148.644
C09707=1183.028,168.590,-56.603,-178.150,6.508,148.644
C09708=1183.033,168.342,-56.582,-178.152,6.506,148.644
C09709=1183.037,168.092,-56.560,-178.155,6.505,148.645
C09710=1183.042,167.844,-56.538,-178.158,6.503,148.645
C09711=1183.046,167.594,-56.516,-178.160,6.501,148.646
C09712=1183.052,167.345,-56.494,-178.163,6.499,148.646
C09713=1183.056,167.096,-56.472,-178.166,6.497,148.646
C09714=1183.061,166.847,-56.450,-178.168,6.496,148.647
C09715=1183.065,166.598,-56.428,-178.171,6.494,148.647
C09716=1183.070,166.349,-56.406,-178.174,6.492,148.647
C09717=1183.075,166.100,-56.384,-178.176,6.490,148.648
C09718=1183.079,165.852,-56.362,-178.179,6.489,148.648
C09719=1183.084,165.603,-56.340,-178.182,6.487,148.648
C09720=1183.089,165.353,-56.318,-178.184,6.486,148.649
C09721=1183.094,165.104,-56.297,-178.187,6.484,148.649
C09722=1183.098,164.855,-56.274,-178.190,6.483,148.650
C09723=1183.103,164.606,-56.253,-178.192,6.481,148.650
C09724=1183.108,164.357,-56.231,-178.195,6.479,148.651
C09725=1183.112,164.108,-56.209,-178.198,6.477,148.651
C09726=1183.117,163.859,-56.187,-178.200,6.476,148.651
C09727=1183.122,163.610,-56.165,-178.203,6.474,148.652
C09728=1183.126,163.362,-56.144,-178.206,6.472,148.652
C09729=1183.131,163.113,-56.122,-178.208,6.470,148.652
C09730=1183.136,162.864,-56.100,-178.211,6.468,148.653
C09731=1183.140,162.615,-56.078,-178.214,6.467,148.653
C09732=1183.145,162.365,-56.057,-178.216,6.465,148.653
C09733=1183.150,162.117,-56.035,-178.219,6.463,148.654
C09734=1183.154,161.867,-56.013,-178.222,6.461,148.654
C09735=1183.159,161.619,-55.991,-178.224,6.460,148.655
C09736=1183.163,161.369,-55.969,-178.227,6.458,148.655
C09737=1183.168,161.121,-55.948,-178.230,6.456,148.655
C09738=1183.173,160.871,-55.927,-178.233,6.454,148.656
C09739=1183.178,160.622,-55.905,-178.235,6.453,148.656
C09740=1183.182,160.373,-55.883,-178.237,6.452,148.656
C09741=1183.187,160.125,-55.861,-178.240,6.450,148.657
C09742=1183.192,159.875,-55.840,-178.243,6.448,148.657
C09743=1183.197,159.626,-55.818,-178.245,6.446,148.658
C09744=1183.202,159.378,-55.797,-178.248,6.445,148.658
C09745=1183.206,159.128,-55.775,-178.251,6.443,148.659
C09746=1183.211,158.859,-55.752,-178.254,6.441,148.659
C09747=1183.216,158.590,-55.729,-178.257,6.440,148.659
C09748=1183.221,158.321,-55.706,-178.260,6.437,148.660
C09749=1183.227,158.053,-55.682,-178.263,6.435,148.660
C09750=1183.230,157.803,-55.661,-178.266,6.434,148.661
C09751=1183.235,157.554,-55.640,-178.268,6.433,148.661
C09752=1183.240,157.306,-55.618,-178.270,6.431,148.661
C09753=1183.245,157.056,-55.597,-178.273,6.429,148.662
C09754=1183.250,156.807,-55.575,-178.276,6.428,148.662
C09755=1183.255,156.558,-55.554,-178.279,6.426,148.663
C09756=1183.259,156.310,-55.533,-178.281,6.424,148.663
C09757=1183.263,156.060,-55.511,-178.284,6.422,148.663
C09758=1183.268,155.811,-55.490,-178.287,6.420,148.664
C09759=1183.273,155.562,-55.468,-178.289,6.419,148.664
C09760=1183.278,155.312,-55.447,-178.292,6.417,148.664
C09761=1183.283,155.064,-55.425,-178.294,6.416,148.665
C09762=1183.287,154.815,-55.405,-178.297,6.414,148.665
C09763=1183.292,154.566,-55.383,-178.300,6.413,148.666
C09764=1183.297,154.316,-55.362,-178.303,6.411,148.666
C09765=1183.301,154.068,-55.340,-178.305,6.409,148.667
C09766=1183.306,153.819,-55.320,-178.308,6.407,148.667
C09767=1183.311,153.570,-55.298,-178.311,6.406,148.667
C09768=1183.316,153.321,-55.277,-178.313,6.404,148.668
C09769=1183.320,153.071,-55.255,-178.316,6.402,148.668
C09770=1183.325,152.822,-55.235,-178.318,6.401,148.668
C09771=1183.330,152.574,-55.213,-178.321,6.399,148.669
C09772=1183.335,152.325,-55.192,-178.324,6.398,148.669
C09773=1183.340,152.075,-55.171,-178.327,6.396,148.670
C09774=1183.343,151.826,-55.150,-178.329,6.395,148.670
C09775=1183.349,151.577,-55.129,-178.332,6.393,148.671
C09776=1183.353,151.328,-55.107,-178.335,6.391,148.671
C09777=1183.358,151.079,-55.087,-178.337,6.389,148.671
C09778=1183.363,150.830,-55.066,-178.340,6.388,148.672
C09779=1183.367,150.581,-55.044,-178.342,6.387,148.672
C09780=1183.372,150.332,-55.023,-178.345,6.385,148.672
C09781=1183.377,150.083,-55.002,-178.348,6.383,148.673
C09782=1183.382,149.834,-54.981,-178.351,6.382,148.673
C09783=1183.386,149.585,-54.960,-178.353,6.380,148.674
C09784=1183.391,149.336,-54.939,-178.356,6.378,148.674
C09785=1183.396,149.086,-54.918,-178.358,6.377,148.675
C09786=1183.400,148.837,-54.897,-178.361,6.375,148.675
C09787=1183.405,148.588,-54.876,-178.364,6.374,148.675
C09788=1183.410,148.339,-54.855,-178.366,6.372,148.676
C09789=1183.415,148.090,-54.834,-178.370,6.370,148.676
C09790=1183.420,147.841,-54.813,-178.372,6.369,148.677
C09791=1183.424,147.592,-54.792,-178.375,6.367,148.677
C09792=1183.429,147.343,-54.771,-178.377,6.366,148.677
C09793=1183.433,147.093,-54.751,-178.380,6.364,148.678
C09794=1183.438,146.844,-54.730,-178.382,6.362,148.678
C09795=1183.443,146.596,-54.709,-178.385,6.361,148.679
C09796=1183.448,146.347,-54.688,-178.388,6.359,148.679
C09797=1183.452,146.098,-54.667,-178.391,6.357,148.680
C09798=1183.457,145.848,-54.646,-178.393,6.357,148.680
C09799=1183.462,145.599,-54.626,-178.396,6.355,148.680
C09800=1183.467,145.350,-54.605,-178.398,6.353,148.681
C09801=1183.471,145.101,-54.585,-178.401,6.351,148.681
C09802=1183.476,144.853,-54.563,-178.404,6.350,148.682
C09803=1183.481,144.604,-54.543,-178.407,6.348,148.682
C09804=1183.486,144.354,-54.522,-178.409,6.347,148.683
C09805=1183.490,144.105,-54.501,-178.412,6.345,148.683
C09806=1183.495,143.855,-54.480,-178.414,6.344,148.683
C09807=1183.499,143.607,-54.460,-178.417,6.342,148.684
C09808=1183.504,143.357,-54.439,-178.420,6.340,148.684
C09809=1183.509,143.108,-54.418,-178.422,6.340,148.685
C09810=1183.514,142.859,-54.397,-178.425,6.338,148.685
C09811=1183.519,142.610,-54.377,-178.428,6.336,148.685
C09812=1183.524,142.361,-54.356,-178.431,6.334,148.686
C09813=1183.528,142.112,-54.336,-178.433,6.332,148.686
C09814=1183.533,141.863,-54.315,-178.435,6.332,148.687
C09815=1183.538,141.614,-54.294,-178.439,6.330,148.687
C09816=1183.542,141.365,-54.274,-178.441,6.328,148.688
C09817=1183.547,141.116,-54.253,-178.444,6.327,148.688
C09818=1183.552,140.867,-54.232,-178.447,6.325,148.688
C09819=1183.556,140.618,-54.212,-178.449,6.324,148.689
C09820=1183.562,140.368,-54.192,-178.451,6.322,148.689
C09821=1183.566,140.119,-54.171,-178.455,6.321,148.690
C09822=1183.571,139.870,-54.151,-178.457,6.319,148.690
C09823=1183.576,139.621,-54.130,-178.460,6.317,148.691
C09824=1183.580,139.372,-54.110,-178.462,6.316,148.691
C09825=1183.585,139.123,-54.089,-178.465,6.315,148.691
C09826=1183.590,138.873,-54.068,-178.468,6.313,148.692
C09827=1183.594,138.624,-54.048,-178.471,6.311,148.692
C09828=1183.599,138.375,-54.028,-178.473,6.310,148.693
C09829=1183.604,138.126,-54.007,-178.475,6.309,148.693
C09830=1183.609,137.877,-53.987,-178.478,6.307,148.694
C09831=1183.614,137.628,-53.967,-178.481,6.306,148.694
C09832=1183.618,137.380,-53.947,-178.484,6.304,148.695
C09833=1183.624,137.130,-53.926,-178.486,6.303,148.695
C09834=1183.628,136.881,-53.906,-178.489,6.301,148.695
C09835=1183.632,136.632,-53.886,-178.492,6.299,148.696
C09836=1183.638,136.382,-53.865,-178.495,6.298,148.696
C09837=1183.642,136.133,-53.845,-178.497,6.297,148.697
C09838=1183.647,135.884,-53.825,-178.500,6.295,148.697
C09839=1183.651,135.635,-53.804,-178.502,6.293,148.698
C09840=1183.656,135.385,-53.785,-178.505,6.292,148.698
C09841=1183.661,135.136,-53.764,-178.508,6.290,148.698
C09842=1183.666,134.888,-53.744,-178.510,6.289,148.699
C09843=1183.671,134.638,-53.724,-178.513,6.288,148.699
C09844=1183.675,134.389,-53.704,-178.516,6.286,148.700
C09845=1183.680,134.140,-53.683,-178.519,6.284,148.700
C09846=1183.685,133.891,-53.663,-178.521,6.284,148.701
C09847=1183.690,133.642,-53.643,-178.524,6.282,148.701
C09848=1183.694,133.393,-53.622,-178.526,6.280,148.701
C09849=1183.700,133.144,-53.603,-178.529,6.278,148.702
C09850=1183.704,132.875,-53.580,-178.532,6.277,148.702
C09851=1183.709,132.606,-53.559,-178.534,6.276,148.703
C09852=1183.715,132.337,-53.537,-178.537,6.275,148.704
C09853=1183.719,132.069,-53.516,-178.540,6.273,148.704
C09854=1183.725,131.820,-53.496,-178.543,6.271,148.704
C09855=1183.729,131.571,-53.476,-178.546,6.270,148.705
C09856=1183.735,131.321,-53.456,-178.549,6.268,148.705
C09857=1183.739,131.072,-53.435,-178.551,6.267,148.706
C09858=1183.744,130.823,-53.416,-178.554,6.265,148.706
C09859=1183.748,130.574,-53.395,-178.557,6.264,148.707
C09860=1183.754,130.325,-53.376,-178.559,6.263,148.707
C09861=1183.758,130.076,-53.356,-178.562,6.261,148.707
C09862=1183.763,129.827,-53.336,-178.564,6.259,148.708
C09863=1183.767,129.578,-53.316,-178.567,6.258,148.709
C09864=1183.773,129.329,-53.296,-178.570,6.257,148.709
C09865=1183.777,129.080,-53.276,-178.572,6.255,148.709
C09866=1183.782,128.830,-53.256,-178.575,6.254,148.710
C09867=1183.787,128.581,-53.237,-178.578,6.252,148.710
C09868=1183.791,128.332,-53.216,-178.580,6.251,148.711
C09869=1183.796,128.083,-53.197,-178.583,6.249,148.711
C09870=1183.801,127.834,-53.177,-178.586,6.248,148.712
C09871=1183.806,127.584,-53.157,-178.588,6.247,148.712
C09872=1183.810,127.335,-53.137,-178.591,6.245,148.713
C09873=1183.815,127.087,-53.117,-178.594,6.244,148.713
C09874=1183.820,126.837,-53.098,-178.596,6.243,148.713
C09875=1183.825,126.587,-53.078,-178.599,6.241,148.714
C09876=1183.829,126.338,-53.058,-178.602,6.240,148.714
C09877=1183.835,126.090,-53.038,-178.604,6.238,148.715
C09878=1183.839,125.840,-53.019,-178.606,6.237,148.715
C09879=1183.844,125.591,-52.998,-178.610,6.235,148.716
C09880=1183.849,125.342,-52.979,-178.612,6.234,148.716
C09881=1183.854,125.093,-52.959,-178.614,6.233,148.717
C09882=1183.859,124.843,-52.940,-178.618,6.231,148.717
C09883=1183.863,124.594,-52.919,-178.620,6.230,148.718
C09884=1183.868,124.345,-52.900,-178.623,6.229,148.718
C09885=1183.873,124.096,-52.880,-178.625,6.227,148.718
C09886=1183.878,123.846,-52.861,-178.628,6.226,148.719
C09887=1183.882,123.598,-52.841,-178.631,6.225,148.719
C09888=1183.887,123.349,-52.822,-178.633,6.223,148.720
C09889=1183.892,123.099,-52.802,-178.636,6.222,148.720
C09890=1183.897,122.850,-52.783,-178.639,6.220,148.721
C09891=1183.902,122.601,-52.763,-178.641,6.219,148.721
C09892=1183.906,122.351,-52.743,-178.644,6.217,148.722
C09893=1183.911,122.103,-52.723,-178.647,6.216,148.722
C09894=1183.915,121.854,-52.704,-178.649,6.215,148.723
C09895=1183.920,121.604,-52.685,-178.652,6.213,148.723
C09896=1183.926,121.355,-52.665,-178.655,6.212,148.724
C09897=1183.930,121.106,-52.646,-178.657,6.211,148.724
C09898=1183.935,120.856,-52.626,-178.660,6.209,148.724
C09899=1183.940,120.607,-52.607,-178.663,6.208,148.725
C09900=1183.944,120.358,-52.588,-178.665,6.207,148.726
C09901=1183.950,120.109,-52.568,-178.668,6.205,148.726
C09902=1183.955,119.859,-52.549,-178.671,6.203,148.726
C09903=1183.959,119.610,-52.528,-178.673,6.203,148.727
C09904=1183.964,119.362,-52.510,-178.676,6.201,148.727
C09905=1183.968,119.112,-52.490,-178.678,6.200,148.728
C09906=1183.973,118.863,-52.470,-178.681,6.199,148.728
C09907=1183.978,118.614,-52.451,-178.684,6.197,148.729
C09908=1183.983,118.364,-52.431,-178.686,6.196,148.729
C09909=1183.988,118.116,-52.413,-178.689,6.194,148.730
C09910=1183.992,117.866,-52.393,-178.692,6.193,148.730
C09911=1183.998,117.617,-52.374,-178.694,6.192,148.731
C09912=1184.002,117.367,-52.355,-178.697,6.190,148.731
C09913=1184.007,117.118,-52.336,-178.700,6.189,148.732
C09914=1184.012,116.869,-52.317,-178.702,6.188,148.732
C09915=1184.017,116.619,-52.297,-178.705,6.186,148.733
C09916=1184.022,116.371,-52.278,-178.708,6.185,148.733
C09917=1184.026,116.121,-52.259,-178.710,6.184,148.734
C09918=1184.032,115.872,-52.239,-178.713,6.182,148.734
C09919=1184.036,115.623,-52.220,-178.715,6.181,148.735
C09920=1184.041,115.374,-52.201,-178.718,6.180,148.735
C09921=1184.046,115.125,-52.181,-178.721,6.178,148.736
C09922=1184.051,114.876,-52.163,-178.724,6.177,148.736
C09923=1184.055,114.626,-52.144,-178.726,6.176,148.736
C09924=1184.061,114.377,-52.124,-178.729,6.174,148.737
C09925=1184.065,114.128,-52.105,-178.732,6.173,148.737
C09926=1184.070,113.879,-52.086,-178.734,6.172,148.738
C09927=1184.074,113.630,-52.067,-178.737,6.171,148.738
C09928=1184.080,113.380,-52.048,-178.740,6.169,148.739
C09929=1184.084,113.131,-52.029,-178.742,6.168,148.739
C09930=1184.089,112.882,-52.010,-178.745,6.167,148.740
C09931=1184.094,112.633,-51.990,-178.748,6.165,148.740
C09932=1184.099,112.383,-51.972,-178.750,6.164,148.741
C09933=1184.103,112.134,-51.953,-178.753,6.163,148.741
C09934=1184.109,111.885,-51.933,-178.756,6.161,148.742
C09935=1184.113,111.636,-51.914,-178.758,6.160,148.742
C09936=1184.118,111.386,-51.896,-178.761,6.159,148.743
C09937=1184.122,111.137,-51.877,-178.763,6.158,148.743
C09938=1184.128,110.888,-51.857,-178.766,6.156,148.744
C09939=1184.132,110.638,-51.839,-178.769,6.155,148.744
C09940=1184.137,110.389,-51.820,-178.771,6.154,148.745
C09941=1184.141,110.140,-51.801,-178.774,6.153,148.745
C09942=1184.147,109.891,-51.782,-178.776,6.152,148.746
C09943=1184.152,109.642,-51.763,-178.779,6.150,148.746
C09944=1184.156,109.392,-51.744,-178.782,6.148,148.747
C09945=1184.161,109.143,-51.726,-178.784,6.148,148.747
C09946=1184.166,108.894,-51.706,-178.787,6.146,148.748
C09947=1184.171,108.645,-51.688,-178.790,6.145,148.748
C09948=1184.176,108.395,-51.669,-178.792,6.144,148.749
C09949=1184.180,108.146,-51.650,-178.795,6.142,148.749
C09950=1184.186,107.897,-51.631,-178.798,6.141,148.750
C09951=1184.190,107.648,-51.612,-178.800,6.139,148.750
C09952=1184.196,107.398,-51.594,-178.803,6.139,148.751
C09953=1184.200,107.150,-51.575,-178.806,6.137,148.751
C09954=1184.206,106.880,-51.555,-178.809,6.136,148.752
C09955=1184.210,106.613,-51.534,-178.811,6.135,148.752
C09956=1184.216,106.344,-51.514,-178.814,6.134,148.753
C09957=1184.220,106.076,-51.494,-178.817,6.132,148.753
C09958=1184.226,105.826,-51.475,-178.820,6.131,148.754
C09959=1184.231,105.578,-51.457,-178.822,6.129,148.754
C09960=1184.236,105.328,-51.438,-178.825,6.128,148.755
C09961=1184.241,105.078,-51.420,-178.828,6.127,148.755
C09962=1184.245,104.829,-51.401,-178.830,6.125,148.756
C09963=1184.250,104.580,-51.382,-178.833,6.125,148.756
C09964=1184.255,104.331,-51.363,-178.836,6.123,148.757
C09965=1184.259,104.081,-51.345,-178.838,6.122,148.757
C09966=1184.264,103.832,-51.326,-178.841,6.121,148.758
C09967=1184.269,103.583,-51.308,-178.843,6.120,148.758
C09968=1184.274,103.333,-51.289,-178.846,6.118,148.759
C09969=1184.279,103.084,-51.270,-178.849,6.117,148.759
C09970=1184.284,102.835,-51.252,-178.851,6.116,148.760
C09971=1184.289,102.586,-51.234,-178.854,6.115,148.760
C09972=1184.294,102.337,-51.215,-178.857,6.114,148.761
C09973=1184.298,102.087,-51.197,-178.859,6.112,148.761
C09974=1184.303,101.839,-51.178,-178.862,6.111,148.762
C09975=1184.308,101.589,-51.159,-178.865,6.110,148.762
C09976=1184.313,101.339,-51.141,-178.867,6.109,148.763
C09977=1184.318,101.090,-51.123,-178.870,6.107,148.763
C09978=1184.322,100.841,-51.104,-178.873,6.107,148.764
C09979=1184.328,100.592,-51.085,-178.875,6.105,148.764
C09980=1184.333,100.342,-51.067,-178.878,6.103,148.765
C09981=1184.337,100.094,-51.049,-178.881,6.103,148.765
C09982=1184.341,99.844,-51.030,-178.883,6.101,148.766
C09983=1184.347,99.594,-51.012,-178.886,6.100,148.766
C09984=1184.352,99.345,-50.994,-178.889,6.099,148.767
C09985=1184.357,99.097,-50.975,-178.891,6.098,148.767
C09986=1184.361,98.847,-50.957,-178.894,6.096,148.768
C09987=1184.366,98.598,-50.939,-178.896,6.096,148.768
C09988=1184.371,98.348,-50.920,-178.899,6.094,148.769
C09989=1184.376,98.099,-50.902,-178.901,6.093,148.769
C09990=1184.381,97.849,-50.884,-178.905,6.092,148.770
C09991=1184.385,97.601,-50.865,-178.907,6.091,148.770
C09992=1184.390,97.351,-50.847,-178.909,6.089,148.771
C09993=1184.395,97.102,-50.829,-178.912,6.089,148.771
C09994=1184.401,96.853,-50.811,-178.915,6.087,148.772
C09995=1184.405,96.603,-50.792,-178.917,6.086,148.773
C09996=1184.410,96.354,-50.774,-178.920,6.085,148.773
//INST
///DATE 2021/06/15 17:24
///ATTR SC,RW,RJ
////FRAME ROBOT
///GROUP1 RB1
NOP
MOVL C00000 V=800.0 PL=0
MOVL C00001 V=800.0 PL=0
MOVL C00002 V=800.0 PL=0
MOVL C00003 V=800.0 PL=0
MOVL C00004 V=800.0 PL=0
MOVL C00005 V=800.0 PL=0
MOVL C00006 V=800.0 PL=0
MOVL C00007 V=800.0 PL=0
MOVL C00008 V=800.0 PL=0
MOVL C00009 V=800.0 PL=0
MOVL C00010 V=800.0 PL=0
MOVL C00011 V=800.0 PL=0
MOVL C00012 V=800.0 PL=0
MOVL C00013 V=800.0 PL=0
MOVL C00014 V=800.0 PL=0
MOVL C00015 V=800.0 PL=0
MOVL C00016 V=800.0 PL=0
MOVL C00017 V=800.0 PL=0
MOVL C00018 V=800.0 PL=0
MOVL C00019 V=800.0 PL=0
MOVL C00020 V=800.0 PL=0
MOVL C00021 V=800.0 PL=0
MOVL C00022 V=800.0 PL=0
MOVL C00023 V=800.0 PL=0
MOVL C00024 V=800.0 PL=0
MOVL C00025 V=800.0 PL=0
MOVL C00026 V=800.0 PL=0
MOVL C00027 V=800.0 PL=0
MOVL C00028 V=800.0 PL=0
MOVL C00029 V=800.0 PL=0
MOVL C00030 V=800.0 PL=0
MOVL C00031 V=800.0 PL=0
MOVL C00032 V=800.0 PL=0
MOVL C00033 V=800.0 PL=0
MOVL C00034 V=800.0 PL=0
MOVL C00035 V=800.0 PL=0
MOVL C00036 V=800.0 PL=0
MOVL C00037 V=800.0 PL=0
MOVL C00038 V=800.0 PL=0
MOVL C00039 V=800.0 PL=0
MOVL C00040 V=800.0 PL=0
MOVL C00041 V=800.0 PL=0
MOVL C00042 V=800.0 PL=0
MOVL C00043 V=800.0 PL=0
MOVL C00044 V=800.0 PL=0
MOVL C00045 V=800.0 PL=0
MOVL C00046 V=800.0 PL=0
MOVL C00047 V=800.0 PL=0
MOVL C00048 V=800.0 PL=0
MOVL C00049 V=800.0 PL=0
MOVL C00050 V=800.0 PL=0
MOVL C00051 V=800.0 PL=0
MOVL C00052 V=800.0 PL=0
MOVL C00053 V=800.0 PL=0
MOVL C00054 V=800.0 PL=0
MOVL C00055 V=800.0 PL=0
MOVL C00056 V=800.0 PL=0
MOVL C00057 V=800.0 PL=0
MOVL C00058 V=800.0 PL=0
MOVL C00059 V=800.0 PL=0
MOVL C00060 V=800.0 PL=0
MOVL C00061 V=800.0 PL=0
MOVL C00062 V=800.0 PL=0
MOVL C00063 V=800.0 PL=0
MOVL C00064 V=800.0 PL=0
MOVL C00065 V=800.0 PL=0
MOVL C00066 V=800.0 PL=0
MOVL C00067 V=800.0 PL=0
MOVL C00068 V=800.0 PL=0
MOVL C00069 V=800.0 PL=0
MOVL C00070 V=800.0 PL=0
MOVL C00071 V=800.0 PL=0
MOVL C00072 V=800.0 PL=0
MOVL C00073 V=800.0 PL=0
MOVL C00074 V=800.0 PL=0
MOVL C00075 V=800.0 PL=0
MOVL C00076 V=800.0 PL=0
MOVL C00077 V=800.0 PL=0
MOVL C00078 V=800.0 PL=0
MOVL C00079 V=800.0 PL=0
MOVL C00080 V=800.0 PL=0
MOVL C00081 V=800.0 PL=0
MOVL C00082 V=800.0 PL=0
MOVL C00083 V=800.0 PL=0
MOVL C00084 V=800.0 PL=0
MOVL C00085 V=800.0 PL=0
MOVL C00086 V=800.0 PL=0
MOVL C00087 V=800.0 PL=0
MOVL C00088 V=800.0 PL=0
MOVL C00089 V=800.0 PL=0
MOVL C00090 V=800.0 PL=0
MOVL C00091 V=800.0 PL=0
MOVL C00092 V=800.0 PL=0
MOVL C00093 V=800.0 PL=0
MOVL C00094 V=800.0 PL=0
MOVL C00095 V=800.0 PL=0
MOVL C00096 V=800.0 PL=0
MOVL C00097 V=800.0 PL=0
MOVL C00098 V=800.0 PL=0
MOVL C00099 V=800.0 PL=0
MOVL C00100 V=800.0 PL=0
MOVL C00101 V=800.0 PL=0
MOVL C00102 V=800.0 PL=0
MOVL C00103 V=800.0 PL=0
MOVL C00104 V=800.0 PL=0
MOVL C00105 V=800.0 PL=0
MOVL C00106 V=800.0 PL=0
MOVL C00107 V=800.0 PL=0
MOVL C00108 V=800.0 PL=0
MOVL C00109 V=800.0 PL=0
MOVL C00110 V=800.0 PL=0
MOVL C00111 V=800.0 PL=0
MOVL C00112 V=800.0 PL=0
MOVL C00113 V=800.0 PL=0
MOVL C00114 V=800.0 PL=0
MOVL C00115 V=800.0 PL=0
MOVL C00116 V=800.0 PL=0
MOVL C00117 V=800.0 PL=0
MOVL C00118 V=800.0 PL=0
MOVL C00119 V=800.0 PL=0
MOVL C00120 V=800.0 PL=0
MOVL C00121 V=800.0 PL=0
MOVL C00122 V=800.0 PL=0
MOVL C00123 V=800.0 PL=0
MOVL C00124 V=800.0 PL=0
MOVL C00125 V=800.0 PL=0
MOVL C00126 V=800.0 PL=0
MOVL C00127 V=800.0 PL=0
MOVL C00128 V=800.0 PL=0
MOVL C00129 V=800.0 PL=0
MOVL C00130 V=800.0 PL=0
MOVL C00131 V=800.0 PL=0
MOVL C00132 V=800.0 PL=0
MOVL C00133 V=800.0 PL=0
MOVL C00134 V=800.0 PL=0
MOVL C00135 V=800.0 PL=0
MOVL C00136 V=800.0 PL=0
MOVL C00137 V=800.0 PL=0
MOVL C00138 V=800.0 PL=0
MOVL C00139 V=800.0 PL=0
MOVL C00140 V=800.0 PL=0
MOVL C00141 V=800.0 PL=0
MOVL C00142 V=800.0 PL=0
MOVL C00143 V=800.0 PL=0
MOVL C00144 V=800.0 PL=0
MOVL C00145 V=800.0 PL=0
MOVL C00146 V=800.0 PL=0
MOVL C00147 V=800.0 PL=0
MOVL C00148 V=800.0 PL=0
MOVL C00149 V=800.0 PL=0
MOVL C00150 V=800.0 PL=0
MOVL C00151 V=800.0 PL=0
MOVL C00152 V=800.0 PL=0
MOVL C00153 V=800.0 PL=0
MOVL C00154 V=800.0 PL=0
MOVL C00155 V=800.0 PL=0
MOVL C00156 V=800.0 PL=0
MOVL C00157 V=800.0 PL=0
MOVL C00158 V=800.0 PL=0
MOVL C00159 V=800.0 PL=0
MOVL C00160 V=800.0 PL=0
MOVL C00161 V=800.0 PL=0
MOVL C00162 V=800.0 PL=0
MOVL C00163 V=800.0 PL=0
MOVL C00164 V=800.0 PL=0
MOVL C00165 V=800.0 PL=0
MOVL C00166 V=800.0 PL=0
MOVL C00167 V=800.0 PL=0
MOVL C00168 V=800.0 PL=0
MOVL C00169 V=800.0 PL=0
MOVL C00170 V=800.0 PL=0
MOVL C00171 V=800.0 PL=0
MOVL C00172 V=800.0 PL=0
MOVL C00173 V=800.0 PL=0
MOVL C00174 V=800.0 PL=0
MOVL C00175 V=800.0 PL=0
MOVL C00176 V=800.0 PL=0
MOVL C00177 V=800.0 PL=0
MOVL C00178 V=800.0 PL=0
MOVL C00179 V=800.0 PL=0
MOVL C00180 V=800.0 PL=0
MOVL C00181 V=800.0 PL=0
MOVL C00182 V=800.0 PL=0
MOVL C00183 V=800.0 PL=0
MOVL C00184 V=800.0 PL=0
MOVL C00185 V=800.0 PL=0
MOVL C00186 V=800.0 PL=0
MOVL C00187 V=800.0 PL=0
MOVL C00188 V=800.0 PL=0
MOVL C00189 V=800.0 PL=0
MOVL C00190 V=800.0 PL=0
MOVL C00191 V=800.0 PL=0
MOVL C00192 V=800.0 PL=0
MOVL C00193 V=800.0 PL=0
MOVL C00194 V=800.0 PL=0
MOVL C00195 V=800.0 PL=0
MOVL C00196 V=800.0 PL=0
MOVL C00197 V=800.0 PL=0
MOVL C00198 V=800.0 PL=0
MOVL C00199 V=800.0 PL=0
MOVL C00200 V=800.0 PL=0
MOVL C00201 V=800.0 PL=0
MOVL C00202 V=800.0 PL=0
MOVL C00203 V=800.0 PL=0
MOVL C00204 V=800.0 PL=0
MOVL C00205 V=800.0 PL=0
MOVL C00206 V=800.0 PL=0
MOVL C00207 V=800.0 PL=0
MOVL C00208 V=800.0 PL=0
MOVL C00209 V=800.0 PL=0
MOVL C00210 V=800.0 PL=0
MOVL C00211 V=800.0 PL=0
MOVL C00212 V=800.0 PL=0
MOVL C00213 V=800.0 PL=0
MOVL C00214 V=800.0 PL=0
MOVL C00215 V=800.0 PL=0
MOVL C00216 V=800.0 PL=0
MOVL C00217 V=800.0 PL=0
MOVL C00218 V=800.0 PL=0
MOVL C00219 V=800.0 PL=0
MOVL C00220 V=800.0 PL=0
MOVL C00221 V=800.0 PL=0
MOVL C00222 V=800.0 PL=0
MOVL C00223 V=800.0 PL=0
MOVL C00224 V=800.0 PL=0
MOVL C00225 V=800.0 PL=0
MOVL C00226 V=800.0 PL=0
MOVL C00227 V=800.0 PL=0
MOVL C00228 V=800.0 PL=0
MOVL C00229 V=800.0 PL=0
MOVL C00230 V=800.0 PL=0
MOVL C00231 V=800.0 PL=0
MOVL C00232 V=800.0 PL=0
MOVL C00233 V=800.0 PL=0
MOVL C00234 V=800.0 PL=0
MOVL C00235 V=800.0 PL=0
MOVL C00236 V=800.0 PL=0
MOVL C00237 V=800.0 PL=0
MOVL C00238 V=800.0 PL=0
MOVL C00239 V=800.0 PL=0
MOVL C00240 V=800.0 PL=0
MOVL C00241 V=800.0 PL=0
MOVL C00242 V=800.0 PL=0
MOVL C00243 V=800.0 PL=0
MOVL C00244 V=800.0 PL=0
MOVL C00245 V=800.0 PL=0
MOVL C00246 V=800.0 PL=0
MOVL C00247 V=800.0 PL=0
MOVL C00248 V=800.0 PL=0
MOVL C00249 V=800.0 PL=0
MOVL C00250 V=800.0 PL=0
MOVL C00251 V=800.0 PL=0
MOVL C00252 V=800.0 PL=0
MOVL C00253 V=800.0 PL=0
MOVL C00254 V=800.0 PL=0
MOVL C00255 V=800.0 PL=0
MOVL C00256 V=800.0 PL=0
MOVL C00257 V=800.0 PL=0
MOVL C00258 V=800.0 PL=0
MOVL C00259 V=800.0 PL=0
MOVL C00260 V=800.0 PL=0
MOVL C00261 V=800.0 PL=0
MOVL C00262 V=800.0 PL=0
MOVL C00263 V=800.0 PL=0
MOVL C00264 V=800.0 PL=0
MOVL C00265 V=800.0 PL=0
MOVL C00266 V=800.0 PL=0
MOVL C00267 V=800.0 PL=0
MOVL C00268 V=800.0 PL=0
MOVL C00269 V=800.0 PL=0
MOVL C00270 V=800.0 PL=0
MOVL C00271 V=800.0 PL=0
MOVL C00272 V=800.0 PL=0
MOVL C00273 V=800.0 PL=0
MOVL C00274 V=800.0 PL=0
MOVL C00275 V=800.0 PL=0
MOVL C00276 V=800.0 PL=0
MOVL C00277 V=800.0 PL=0
MOVL C00278 V=800.0 PL=0
MOVL C00279 V=800.0 PL=0
MOVL C00280 V=800.0 PL=0
MOVL C00281 V=800.0 PL=0
MOVL C00282 V=800.0 PL=0
MOVL C00283 V=800.0 PL=0
MOVL C00284 V=800.0 PL=0
MOVL C00285 V=800.0 PL=0
MOVL C00286 V=800.0 PL=0
MOVL C00287 V=800.0 PL=0
MOVL C00288 V=800.0 PL=0
MOVL C00289 V=800.0 PL=0
MOVL C00290 V=800.0 PL=0
MOVL C00291 V=800.0 PL=0
MOVL C00292 V=800.0 PL=0
MOVL C00293 V=800.0 PL=0
MOVL C00294 V=800.0 PL=0
MOVL C00295 V=800.0 PL=0
MOVL C00296 V=800.0 PL=0
MOVL C00297 V=800.0 PL=0
MOVL C00298 V=800.0 PL=0
MOVL C00299 V=800.0 PL=0
MOVL C00300 V=800.0 PL=0
MOVL C00301 V=800.0 PL=0
MOVL C00302 V=800.0 PL=0
MOVL C00303 V=800.0 PL=0
MOVL C00304 V=800.0 PL=0
MOVL C00305 V=800.0 PL=0
MOVL C00306 V=800.0 PL=0
MOVL C00307 V=800.0 PL=0
MOVL C00308 V=800.0 PL=0
MOVL C00309 V=800.0 PL=0
MOVL C00310 V=800.0 PL=0
MOVL C00311 V=800.0 PL=0
MOVL C00312 V=800.0 PL=0
MOVL C00313 V=800.0 PL=0
MOVL C00314 V=800.0 PL=0
MOVL C00315 V=800.0 PL=0
MOVL C00316 V=800.0 PL=0
MOVL C00317 V=800.0 PL=0
MOVL C00318 V=800.0 PL=0
MOVL C00319 V=800.0 PL=0
MOVL C00320 V=800.0 PL=0
MOVL C00321 V=800.0 PL=0
MOVL C00322 V=800.0 PL=0
MOVL C00323 V=800.0 PL=0
MOVL C00324 V=800.0 PL=0
MOVL C00325 V=800.0 PL=0
MOVL C00326 V=800.0 PL=0
MOVL C00327 V=800.0 PL=0
MOVL C00328 V=800.0 PL=0
MOVL C00329 V=800.0 PL=0
MOVL C00330 V=800.0 PL=0
MOVL C00331 V=800.0 PL=0
MOVL C00332 V=800.0 PL=0
MOVL C00333 V=800.0 PL=0
MOVL C00334 V=800.0 PL=0
MOVL C00335 V=800.0 PL=0
MOVL C00336 V=800.0 PL=0
MOVL C00337 V=800.0 PL=0
MOVL C00338 V=800.0 PL=0
MOVL C00339 V=800.0 PL=0
MOVL C00340 V=800.0 PL=0
MOVL C00341 V=800.0 PL=0
MOVL C00342 V=800.0 PL=0
MOVL C00343 V=800.0 PL=0
MOVL C00344 V=800.0 PL=0
MOVL C00345 V=800.0 PL=0
MOVL C00346 V=800.0 PL=0
MOVL C00347 V=800.0 PL=0
MOVL C00348 V=800.0 PL=0
MOVL C00349 V=800.0 PL=0
MOVL C00350 V=800.0 PL=0
MOVL C00351 V=800.0 PL=0
MOVL C00352 V=800.0 PL=0
MOVL C00353 V=800.0 PL=0
MOVL C00354 V=800.0 PL=0
MOVL C00355 V=800.0 PL=0
MOVL C00356 V=800.0 PL=0
MOVL C00357 V=800.0 PL=0
MOVL C00358 V=800.0 PL=0
MOVL C00359 V=800.0 PL=0
MOVL C00360 V=800.0 PL=0
MOVL C00361 V=800.0 PL=0
MOVL C00362 V=800.0 PL=0
MOVL C00363 V=800.0 PL=0
MOVL C00364 V=800.0 PL=0
MOVL C00365 V=800.0 PL=0
MOVL C00366 V=800.0 PL=0
MOVL C00367 V=800.0 PL=0
MOVL C00368 V=800.0 PL=0
MOVL C00369 V=800.0 PL=0
MOVL C00370 V=800.0 PL=0
MOVL C00371 V=800.0 PL=0
MOVL C00372 V=800.0 PL=0
MOVL C00373 V=800.0 PL=0
MOVL C00374 V=800.0 PL=0
MOVL C00375 V=800.0 PL=0
MOVL C00376 V=800.0 PL=0
MOVL C00377 V=800.0 PL=0
MOVL C00378 V=800.0 PL=0
MOVL C00379 V=800.0 PL=0
MOVL C00380 V=800.0 PL=0
MOVL C00381 V=800.0 PL=0
MOVL C00382 V=800.0 PL=0
MOVL C00383 V=800.0 PL=0
MOVL C00384 V=800.0 PL=0
MOVL C00385 V=800.0 PL=0
MOVL C00386 V=800.0 PL=0
MOVL C00387 V=800.0 PL=0
MOVL C00388 V=800.0 PL=0
MOVL C00389 V=800.0 PL=0
MOVL C00390 V=800.0 PL=0
MOVL C00391 V=800.0 PL=0
MOVL C00392 V=800.0 PL=0
MOVL C00393 V=800.0 PL=0
MOVL C00394 V=800.0 PL=0
MOVL C00395 V=800.0 PL=0
MOVL C00396 V=800.0 PL=0
MOVL C00397 V=800.0 PL=0
MOVL C00398 V=800.0 PL=0
MOVL C00399 V=800.0 PL=0
MOVL C00400 V=800.0 PL=0
MOVL C00401 V=800.0 PL=0
MOVL C00402 V=800.0 PL=0
MOVL C00403 V=800.0 PL=0
MOVL C00404 V=800.0 PL=0
MOVL C00405 V=800.0 PL=0
MOVL C00406 V=800.0 PL=0
MOVL C00407 V=800.0 PL=0
MOVL C00408 V=800.0 PL=0
MOVL C00409 V=800.0 PL=0
MOVL C00410 V=800.0 PL=0
MOVL C00411 V=800.0 PL=0
MOVL C00412 V=800.0 PL=0
MOVL C00413 V=800.0 PL=0
MOVL C00414 V=800.0 PL=0
MOVL C00415 V=800.0 PL=0
MOVL C00416 V=800.0 PL=0
MOVL C00417 V=800.0 PL=0
MOVL C00418 V=800.0 PL=0
MOVL C00419 V=800.0 PL=0
MOVL C00420 V=800.0 PL=0
MOVL C00421 V=800.0 PL=0
MOVL C00422 V=800.0 PL=0
MOVL C00423 V=800.0 PL=0
MOVL C00424 V=800.0 PL=0
MOVL C00425 V=800.0 PL=0
MOVL C00426 V=800.0 PL=0
MOVL C00427 V=800.0 PL=0
MOVL C00428 V=800.0 PL=0
MOVL C00429 V=800.0 PL=0
MOVL C00430 V=800.0 PL=0
MOVL C00431 V=800.0 PL=0
MOVL C00432 V=800.0 PL=0
MOVL C00433 V=800.0 PL=0
MOVL C00434 V=800.0 PL=0
MOVL C00435 V=800.0 PL=0
MOVL C00436 V=800.0 PL=0
MOVL C00437 V=800.0 PL=0
MOVL C00438 V=800.0 PL=0
MOVL C00439 V=800.0 PL=0
MOVL C00440 V=800.0 PL=0
MOVL C00441 V=800.0 PL=0
MOVL C00442 V=800.0 PL=0
MOVL C00443 V=800.0 PL=0
MOVL C00444 V=800.0 PL=0
MOVL C00445 V=800.0 PL=0
MOVL C00446 V=800.0 PL=0
MOVL C00447 V=800.0 PL=0
MOVL C00448 V=800.0 PL=0
MOVL C00449 V=800.0 PL=0
MOVL C00450 V=800.0 PL=0
MOVL C00451 V=800.0 PL=0
MOVL C00452 V=800.0 PL=0
MOVL C00453 V=800.0 PL=0
MOVL C00454 V=800.0 PL=0
MOVL C00455 V=800.0 PL=0
MOVL C00456 V=800.0 PL=0
MOVL C00457 V=800.0 PL=0
MOVL C00458 V=800.0 PL=0
MOVL C00459 V=800.0 PL=0
MOVL C00460 V=800.0 PL=0
MOVL C00461 V=800.0 PL=0
MOVL C00462 V=800.0 PL=0
MOVL C00463 V=800.0 PL=0
MOVL C00464 V=800.0 PL=0
MOVL C00465 V=800.0 PL=0
MOVL C00466 V=800.0 PL=0
MOVL C00467 V=800.0 PL=0
MOVL C00468 V=800.0 PL=0
MOVL C00469 V=800.0 PL=0
MOVL C00470 V=800.0 PL=0
MOVL C00471 V=800.0 PL=0
MOVL C00472 V=800.0 PL=0
MOVL C00473 V=800.0 PL=0
MOVL C00474 V=800.0 PL=0
MOVL C00475 V=800.0 PL=0
MOVL C00476 V=800.0 PL=0
MOVL C00477 V=800.0 PL=0
MOVL C00478 V=800.0 PL=0
MOVL C00479 V=800.0 PL=0
MOVL C00480 V=800.0 PL=0
MOVL C00481 V=800.0 PL=0
MOVL C00482 V=800.0 PL=0
MOVL C00483 V=800.0 PL=0
MOVL C00484 V=800.0 PL=0
MOVL C00485 V=800.0 PL=0
MOVL C00486 V=800.0 PL=0
MOVL C00487 V=800.0 PL=0
MOVL C00488 V=800.0 PL=0
MOVL C00489 V=800.0 PL=0
MOVL C00490 V=800.0 PL=0
MOVL C00491 V=800.0 PL=0
MOVL C00492 V=800.0 PL=0
MOVL C00493 V=800.0 PL=0
MOVL C00494 V=800.0 PL=0
MOVL C00495 V=800.0 PL=0
MOVL C00496 V=800.0 PL=0
MOVL C00497 V=800.0 PL=0
MOVL C00498 V=800.0 PL=0
MOVL C00499 V=800.0 PL=0
MOVL C00500 V=800.0 PL=0
MOVL C00501 V=800.0 PL=0
MOVL C00502 V=800.0 PL=0
MOVL C00503 V=800.0 PL=0
MOVL C00504 V=800.0 PL=0
MOVL C00505 V=800.0 PL=0
MOVL C00506 V=800.0 PL=0
MOVL C00507 V=800.0 PL=0
MOVL C00508 V=800.0 PL=0
MOVL C00509 V=800.0 PL=0
MOVL C00510 V=800.0 PL=0
MOVL C00511 V=800.0 PL=0
MOVL C00512 V=800.0 PL=0
MOVL C00513 V=800.0 PL=0
MOVL C00514 V=800.0 PL=0
MOVL C00515 V=800.0 PL=0
MOVL C00516 V=800.0 PL=0
MOVL C00517 V=800.0 PL=0
MOVL C00518 V=800.0 PL=0
MOVL C00519 V=800.0 PL=0
MOVL C00520 V=800.0 PL=0
MOVL C00521 V=800.0 PL=0
MOVL C00522 V=800.0 PL=0
MOVL C00523 V=800.0 PL=0
MOVL C00524 V=800.0 PL=0
MOVL C00525 V=800.0 PL=0
MOVL C00526 V=800.0 PL=0
MOVL C00527 V=800.0 PL=0
MOVL C00528 V=800.0 PL=0
MOVL C00529 V=800.0 PL=0
MOVL C00530 V=800.0 PL=0
MOVL C00531 V=800.0 PL=0
MOVL C00532 V=800.0 PL=0
MOVL C00533 V=800.0 PL=0
MOVL C00534 V=800.0 PL=0
MOVL C00535 V=800.0 PL=0
MOVL C00536 V=800.0 PL=0
MOVL C00537 V=800.0 PL=0
MOVL C00538 V=800.0 PL=0
MOVL C00539 V=800.0 PL=0
MOVL C00540 V=800.0 PL=0
MOVL C00541 V=800.0 PL=0
MOVL C00542 V=800.0 PL=0
MOVL C00543 V=800.0 PL=0
MOVL C00544 V=800.0 PL=0
MOVL C00545 V=800.0 PL=0
MOVL C00546 V=800.0 PL=0
MOVL C00547 V=800.0 PL=0
MOVL C00548 V=800.0 PL=0
MOVL C00549 V=800.0 PL=0
MOVL C00550 V=800.0 PL=0
MOVL C00551 V=800.0 PL=0
MOVL C00552 V=800.0 PL=0
MOVL C00553 V=800.0 PL=0
MOVL C00554 V=800.0 PL=0
MOVL C00555 V=800.0 PL=0
MOVL C00556 V=800.0 PL=0
MOVL C00557 V=800.0 PL=0
MOVL C00558 V=800.0 PL=0
MOVL C00559 V=800.0 PL=0
MOVL C00560 V=800.0 PL=0
MOVL C00561 V=800.0 PL=0
MOVL C00562 V=800.0 PL=0
MOVL C00563 V=800.0 PL=0
MOVL C00564 V=800.0 PL=0
MOVL C00565 V=800.0 PL=0
MOVL C00566 V=800.0 PL=0
MOVL C00567 V=800.0 PL=0
MOVL C00568 V=800.0 PL=0
MOVL C00569 V=800.0 PL=0
MOVL C00570 V=800.0 PL=0
MOVL C00571 V=800.0 PL=0
MOVL C00572 V=800.0 PL=0
MOVL C00573 V=800.0 PL=0
MOVL C00574 V=800.0 PL=0
MOVL C00575 V=800.0 PL=0
MOVL C00576 V=800.0 PL=0
MOVL C00577 V=800.0 PL=0
MOVL C00578 V=800.0 PL=0
MOVL C00579 V=800.0 PL=0
MOVL C00580 V=800.0 PL=0
MOVL C00581 V=800.0 PL=0
MOVL C00582 V=800.0 PL=0
MOVL C00583 V=800.0 PL=0
MOVL C00584 V=800.0 PL=0
MOVL C00585 V=800.0 PL=0
MOVL C00586 V=800.0 PL=0
MOVL C00587 V=800.0 PL=0
MOVL C00588 V=800.0 PL=0
MOVL C00589 V=800.0 PL=0
MOVL C00590 V=800.0 PL=0
MOVL C00591 V=800.0 PL=0
MOVL C00592 V=800.0 PL=0
MOVL C00593 V=800.0 PL=0
MOVL C00594 V=800.0 PL=0
MOVL C00595 V=800.0 PL=0
MOVL C00596 V=800.0 PL=0
MOVL C00597 V=800.0 PL=0
MOVL C00598 V=800.0 PL=0
MOVL C00599 V=800.0 PL=0
MOVL C00600 V=800.0 PL=0
MOVL C00601 V=800.0 PL=0
MOVL C00602 V=800.0 PL=0
MOVL C00603 V=800.0 PL=0
MOVL C00604 V=800.0 PL=0
MOVL C00605 V=800.0 PL=0
MOVL C00606 V=800.0 PL=0
MOVL C00607 V=800.0 PL=0
MOVL C00608 V=800.0 PL=0
MOVL C00609 V=800.0 PL=0
MOVL C00610 V=800.0 PL=0
MOVL C00611 V=800.0 PL=0
MOVL C00612 V=800.0 PL=0
MOVL C00613 V=800.0 PL=0
MOVL C00614 V=800.0 PL=0
MOVL C00615 V=800.0 PL=0
MOVL C00616 V=800.0 PL=0
MOVL C00617 V=800.0 PL=0
MOVL C00618 V=800.0 PL=0
MOVL C00619 V=800.0 PL=0
MOVL C00620 V=800.0 PL=0
MOVL C00621 V=800.0 PL=0
MOVL C00622 V=800.0 PL=0
MOVL C00623 V=800.0 PL=0
MOVL C00624 V=800.0 PL=0
MOVL C00625 V=800.0 PL=0
MOVL C00626 V=800.0 PL=0
MOVL C00627 V=800.0 PL=0
MOVL C00628 V=800.0 PL=0
MOVL C00629 V=800.0 PL=0
MOVL C00630 V=800.0 PL=0
MOVL C00631 V=800.0 PL=0
MOVL C00632 V=800.0 PL=0
MOVL C00633 V=800.0 PL=0
MOVL C00634 V=800.0 PL=0
MOVL C00635 V=800.0 PL=0
MOVL C00636 V=800.0 PL=0
MOVL C00637 V=800.0 PL=0
MOVL C00638 V=800.0 PL=0
MOVL C00639 V=800.0 PL=0
MOVL C00640 V=800.0 PL=0
MOVL C00641 V=800.0 PL=0
MOVL C00642 V=800.0 PL=0
MOVL C00643 V=800.0 PL=0
MOVL C00644 V=800.0 PL=0
MOVL C00645 V=800.0 PL=0
MOVL C00646 V=800.0 PL=0
MOVL C00647 V=800.0 PL=0
MOVL C00648 V=800.0 PL=0
MOVL C00649 V=800.0 PL=0
MOVL C00650 V=800.0 PL=0
MOVL C00651 V=800.0 PL=0
MOVL C00652 V=800.0 PL=0
MOVL C00653 V=800.0 PL=0
MOVL C00654 V=800.0 PL=0
MOVL C00655 V=800.0 PL=0
MOVL C00656 V=800.0 PL=0
MOVL C00657 V=800.0 PL=0
MOVL C00658 V=800.0 PL=0
MOVL C00659 V=800.0 PL=0
MOVL C00660 V=800.0 PL=0
MOVL C00661 V=800.0 PL=0
MOVL C00662 V=800.0 PL=0
MOVL C00663 V=800.0 PL=0
MOVL C00664 V=800.0 PL=0
MOVL C00665 V=800.0 PL=0
MOVL C00666 V=800.0 PL=0
MOVL C00667 V=800.0 PL=0
MOVL C00668 V=800.0 PL=0
MOVL C00669 V=800.0 PL=0
MOVL C00670 V=800.0 PL=0
MOVL C00671 V=800.0 PL=0
MOVL C00672 V=800.0 PL=0
MOVL C00673 V=800.0 PL=0
MOVL C00674 V=800.0 PL=0
MOVL C00675 V=800.0 PL=0
MOVL C00676 V=800.0 PL=0
MOVL C00677 V=800.0 PL=0
MOVL C00678 V=800.0 PL=0
MOVL C00679 V=800.0 PL=0
MOVL C00680 V=800.0 PL=0
MOVL C00681 V=800.0 PL=0
MOVL C00682 V=800.0 PL=0
MOVL C00683 V=800.0 PL=0
MOVL C00684 V=800.0 PL=0
MOVL C00685 V=800.0 PL=0
MOVL C00686 V=800.0 PL=0
MOVL C00687 V=800.0 PL=0
MOVL C00688 V=800.0 PL=0
MOVL C00689 V=800.0 PL=0
MOVL C00690 V=800.0 PL=0
MOVL C00691 V=800.0 PL=0
MOVL C00692 V=800.0 PL=0
MOVL C00693 V=800.0 PL=0
MOVL C00694 V=800.0 PL=0
MOVL C00695 V=800.0 PL=0
MOVL C00696 V=800.0 PL=0
MOVL C00697 V=800.0 PL=0
MOVL C00698 V=800.0 PL=0
MOVL C00699 V=800.0 PL=0
MOVL C00700 V=800.0 PL=0
MOVL C00701 V=800.0 PL=0
MOVL C00702 V=800.0 PL=0
MOVL C00703 V=800.0 PL=0
MOVL C00704 V=800.0 PL=0
MOVL C00705 V=800.0 PL=0
MOVL C00706 V=800.0 PL=0
MOVL C00707 V=800.0 PL=0
MOVL C00708 V=800.0 PL=0
MOVL C00709 V=800.0 PL=0
MOVL C00710 V=800.0 PL=0
MOVL C00711 V=800.0 PL=0
MOVL C00712 V=800.0 PL=0
MOVL C00713 V=800.0 PL=0
MOVL C00714 V=800.0 PL=0
MOVL C00715 V=800.0 PL=0
MOVL C00716 V=800.0 PL=0
MOVL C00717 V=800.0 PL=0
MOVL C00718 V=800.0 PL=0
MOVL C00719 V=800.0 PL=0
MOVL C00720 V=800.0 PL=0
MOVL C00721 V=800.0 PL=0
MOVL C00722 V=800.0 PL=0
MOVL C00723 V=800.0 PL=0
MOVL C00724 V=800.0 PL=0
MOVL C00725 V=800.0 PL=0
MOVL C00726 V=800.0 PL=0
MOVL C00727 V=800.0 PL=0
MOVL C00728 V=800.0 PL=0
MOVL C00729 V=800.0 PL=0
MOVL C00730 V=800.0 PL=0
MOVL C00731 V=800.0 PL=0
MOVL C00732 V=800.0 PL=0
MOVL C00733 V=800.0 PL=0
MOVL C00734 V=800.0 PL=0
MOVL C00735 V=800.0 PL=0
MOVL C00736 V=800.0 PL=0
MOVL C00737 V=800.0 PL=0
MOVL C00738 V=800.0 PL=0
MOVL C00739 V=800.0 PL=0
MOVL C00740 V=800.0 PL=0
MOVL C00741 V=800.0 PL=0
MOVL C00742 V=800.0 PL=0
MOVL C00743 V=800.0 PL=0
MOVL C00744 V=800.0 PL=0
MOVL C00745 V=800.0 PL=0
MOVL C00746 V=800.0 PL=0
MOVL C00747 V=800.0 PL=0
MOVL C00748 V=800.0 PL=0
MOVL C00749 V=800.0 PL=0
MOVL C00750 V=800.0 PL=0
MOVL C00751 V=800.0 PL=0
MOVL C00752 V=800.0 PL=0
MOVL C00753 V=800.0 PL=0
MOVL C00754 V=800.0 PL=0
MOVL C00755 V=800.0 PL=0
MOVL C00756 V=800.0 PL=0
MOVL C00757 V=800.0 PL=0
MOVL C00758 V=800.0 PL=0
MOVL C00759 V=800.0 PL=0
MOVL C00760 V=800.0 PL=0
MOVL C00761 V=800.0 PL=0
MOVL C00762 V=800.0 PL=0
MOVL C00763 V=800.0 PL=0
MOVL C00764 V=800.0 PL=0
MOVL C00765 V=800.0 PL=0
MOVL C00766 V=800.0 PL=0
MOVL C00767 V=800.0 PL=0
MOVL C00768 V=800.0 PL=0
MOVL C00769 V=800.0 PL=0
MOVL C00770 V=800.0 PL=0
MOVL C00771 V=800.0 PL=0
MOVL C00772 V=800.0 PL=0
MOVL C00773 V=800.0 PL=0
MOVL C00774 V=800.0 PL=0
MOVL C00775 V=800.0 PL=0
MOVL C00776 V=800.0 PL=0
MOVL C00777 V=800.0 PL=0
MOVL C00778 V=800.0 PL=0
MOVL C00779 V=800.0 PL=0
MOVL C00780 V=800.0 PL=0
MOVL C00781 V=800.0 PL=0
MOVL C00782 V=800.0 PL=0
MOVL C00783 V=800.0 PL=0
MOVL C00784 V=800.0 PL=0
MOVL C00785 V=800.0 PL=0
MOVL C00786 V=800.0 PL=0
MOVL C00787 V=800.0 PL=0
MOVL C00788 V=800.0 PL=0
MOVL C00789 V=800.0 PL=0
MOVL C00790 V=800.0 PL=0
MOVL C00791 V=800.0 PL=0
MOVL C00792 V=800.0 PL=0
MOVL C00793 V=800.0 PL=0
MOVL C00794 V=800.0 PL=0
MOVL C00795 V=800.0 PL=0
MOVL C00796 V=800.0 PL=0
MOVL C00797 V=800.0 PL=0
MOVL C00798 V=800.0 PL=0
MOVL C00799 V=800.0 PL=0
MOVL C00800 V=800.0 PL=0
MOVL C00801 V=800.0 PL=0
MOVL C00802 V=800.0 PL=0
MOVL C00803 V=800.0 PL=0
MOVL C00804 V=800.0 PL=0
MOVL C00805 V=800.0 PL=0
MOVL C00806 V=800.0 PL=0
MOVL C00807 V=800.0 PL=0
MOVL C00808 V=800.0 PL=0
MOVL C00809 V=800.0 PL=0
MOVL C00810 V=800.0 PL=0
MOVL C00811 V=800.0 PL=0
MOVL C00812 V=800.0 PL=0
MOVL C00813 V=800.0 PL=0
MOVL C00814 V=800.0 PL=0
MOVL C00815 V=800.0 PL=0
MOVL C00816 V=800.0 PL=0
MOVL C00817 V=800.0 PL=0
MOVL C00818 V=800.0 PL=0
MOVL C00819 V=800.0 PL=0
MOVL C00820 V=800.0 PL=0
MOVL C00821 V=800.0 PL=0
MOVL C00822 V=800.0 PL=0
MOVL C00823 V=800.0 PL=0
MOVL C00824 V=800.0 PL=0
MOVL C00825 V=800.0 PL=0
MOVL C00826 V=800.0 PL=0
MOVL C00827 V=800.0 PL=0
MOVL C00828 V=800.0 PL=0
MOVL C00829 V=800.0 PL=0
MOVL C00830 V=800.0 PL=0
MOVL C00831 V=800.0 PL=0
MOVL C00832 V=800.0 PL=0
MOVL C00833 V=800.0 PL=0
MOVL C00834 V=800.0 PL=0
MOVL C00835 V=800.0 PL=0
MOVL C00836 V=800.0 PL=0
MOVL C00837 V=800.0 PL=0
MOVL C00838 V=800.0 PL=0
MOVL C00839 V=800.0 PL=0
MOVL C00840 V=800.0 PL=0
MOVL C00841 V=800.0 PL=0
MOVL C00842 V=800.0 PL=0
MOVL C00843 V=800.0 PL=0
MOVL C00844 V=800.0 PL=0
MOVL C00845 V=800.0 PL=0
MOVL C00846 V=800.0 PL=0
MOVL C00847 V=800.0 PL=0
MOVL C00848 V=800.0 PL=0
MOVL C00849 V=800.0 PL=0
MOVL C00850 V=800.0 PL=0
MOVL C00851 V=800.0 PL=0
MOVL C00852 V=800.0 PL=0
MOVL C00853 V=800.0 PL=0
MOVL C00854 V=800.0 PL=0
MOVL C00855 V=800.0 PL=0
MOVL C00856 V=800.0 PL=0
MOVL C00857 V=800.0 PL=0
MOVL C00858 V=800.0 PL=0
MOVL C00859 V=800.0 PL=0
MOVL C00860 V=800.0 PL=0
MOVL C00861 V=800.0 PL=0
MOVL C00862 V=800.0 PL=0
MOVL C00863 V=800.0 PL=0
MOVL C00864 V=800.0 PL=0
MOVL C00865 V=800.0 PL=0
MOVL C00866 V=800.0 PL=0
MOVL C00867 V=800.0 PL=0
MOVL C00868 V=800.0 PL=0
MOVL C00869 V=800.0 PL=0
MOVL C00870 V=800.0 PL=0
MOVL C00871 V=800.0 PL=0
MOVL C00872 V=800.0 PL=0
MOVL C00873 V=800.0 PL=0
MOVL C00874 V=800.0 PL=0
MOVL C00875 V=800.0 PL=0
MOVL C00876 V=800.0 PL=0
MOVL C00877 V=800.0 PL=0
MOVL C00878 V=800.0 PL=0
MOVL C00879 V=800.0 PL=0
MOVL C00880 V=800.0 PL=0
MOVL C00881 V=800.0 PL=0
MOVL C00882 V=800.0 PL=0
MOVL C00883 V=800.0 PL=0
MOVL C00884 V=800.0 PL=0
MOVL C00885 V=800.0 PL=0
MOVL C00886 V=800.0 PL=0
MOVL C00887 V=800.0 PL=0
MOVL C00888 V=800.0 PL=0
MOVL C00889 V=800.0 PL=0
MOVL C00890 V=800.0 PL=0
MOVL C00891 V=800.0 PL=0
MOVL C00892 V=800.0 PL=0
MOVL C00893 V=800.0 PL=0
MOVL C00894 V=800.0 PL=0
MOVL C00895 V=800.0 PL=0
MOVL C00896 V=800.0 PL=0
MOVL C00897 V=800.0 PL=0
MOVL C00898 V=800.0 PL=0
MOVL C00899 V=800.0 PL=0
MOVL C00900 V=800.0 PL=0
MOVL C00901 V=800.0 PL=0
MOVL C00902 V=800.0 PL=0
MOVL C00903 V=800.0 PL=0
MOVL C00904 V=800.0 PL=0
MOVL C00905 V=800.0 PL=0
MOVL C00906 V=800.0 PL=0
MOVL C00907 V=800.0 PL=0
MOVL C00908 V=800.0 PL=0
MOVL C00909 V=800.0 PL=0
MOVL C00910 V=800.0 PL=0
MOVL C00911 V=800.0 PL=0
MOVL C00912 V=800.0 PL=0
MOVL C00913 V=800.0 PL=0
MOVL C00914 V=800.0 PL=0
MOVL C00915 V=800.0 PL=0
MOVL C00916 V=800.0 PL=0
MOVL C00917 V=800.0 PL=0
MOVL C00918 V=800.0 PL=0
MOVL C00919 V=800.0 PL=0
MOVL C00920 V=800.0 PL=0
MOVL C00921 V=800.0 PL=0
MOVL C00922 V=800.0 PL=0
MOVL C00923 V=800.0 PL=0
MOVL C00924 V=800.0 PL=0
MOVL C00925 V=800.0 PL=0
MOVL C00926 V=800.0 PL=0
MOVL C00927 V=800.0 PL=0
MOVL C00928 V=800.0 PL=0
MOVL C00929 V=800.0 PL=0
MOVL C00930 V=800.0 PL=0
MOVL C00931 V=800.0 PL=0
MOVL C00932 V=800.0 PL=0
MOVL C00933 V=800.0 PL=0
MOVL C00934 V=800.0 PL=0
MOVL C00935 V=800.0 PL=0
MOVL C00936 V=800.0 PL=0
MOVL C00937 V=800.0 PL=0
MOVL C00938 V=800.0 PL=0
MOVL C00939 V=800.0 PL=0
MOVL C00940 V=800.0 PL=0
MOVL C00941 V=800.0 PL=0
MOVL C00942 V=800.0 PL=0
MOVL C00943 V=800.0 PL=0
MOVL C00944 V=800.0 PL=0
MOVL C00945 V=800.0 PL=0
MOVL C00946 V=800.0 PL=0
MOVL C00947 V=800.0 PL=0
MOVL C00948 V=800.0 PL=0
MOVL C00949 V=800.0 PL=0
MOVL C00950 V=800.0 PL=0
MOVL C00951 V=800.0 PL=0
MOVL C00952 V=800.0 PL=0
MOVL C00953 V=800.0 PL=0
MOVL C00954 V=800.0 PL=0
MOVL C00955 V=800.0 PL=0
MOVL C00956 V=800.0 PL=0
MOVL C00957 V=800.0 PL=0
MOVL C00958 V=800.0 PL=0
MOVL C00959 V=800.0 PL=0
MOVL C00960 V=800.0 PL=0
MOVL C00961 V=800.0 PL=0
MOVL C00962 V=800.0 PL=0
MOVL C00963 V=800.0 PL=0
MOVL C00964 V=800.0 PL=0
MOVL C00965 V=800.0 PL=0
MOVL C00966 V=800.0 PL=0
MOVL C00967 V=800.0 PL=0
MOVL C00968 V=800.0 PL=0
MOVL C00969 V=800.0 PL=0
MOVL C00970 V=800.0 PL=0
MOVL C00971 V=800.0 PL=0
MOVL C00972 V=800.0 PL=0
MOVL C00973 V=800.0 PL=0
MOVL C00974 V=800.0 PL=0
MOVL C00975 V=800.0 PL=0
MOVL C00976 V=800.0 PL=0
MOVL C00977 V=800.0 PL=0
MOVL C00978 V=800.0 PL=0
MOVL C00979 V=800.0 PL=0
MOVL C00980 V=800.0 PL=0
MOVL C00981 V=800.0 PL=0
MOVL C00982 V=800.0 PL=0
MOVL C00983 V=800.0 PL=0
MOVL C00984 V=800.0 PL=0
MOVL C00985 V=800.0 PL=0
MOVL C00986 V=800.0 PL=0
MOVL C00987 V=800.0 PL=0
MOVL C00988 V=800.0 PL=0
MOVL C00989 V=800.0 PL=0
MOVL C00990 V=800.0 PL=0
MOVL C00991 V=800.0 PL=0
MOVL C00992 V=800.0 PL=0
MOVL C00993 V=800.0 PL=0
MOVL C00994 V=800.0 PL=0
MOVL C00995 V=800.0 PL=0
MOVL C00996 V=800.0 PL=0
MOVL C00997 V=800.0 PL=0
MOVL C00998 V=800.0 PL=0
MOVL C00999 V=800.0 PL=0
MOVL C01000 V=800.0 PL=0
MOVL C01001 V=800.0 PL=0
MOVL C01002 V=800.0 PL=0
MOVL C01003 V=800.0 PL=0
MOVL C01004 V=800.0 PL=0
MOVL C01005 V=800.0 PL=0
MOVL C01006 V=800.0 PL=0
MOVL C01007 V=800.0 PL=0
MOVL C01008 V=800.0 PL=0
MOVL C01009 V=800.0 PL=0
MOVL C01010 V=800.0 PL=0
MOVL C01011 V=800.0 PL=0
MOVL C01012 V=800.0 PL=0
MOVL C01013 V=800.0 PL=0
MOVL C01014 V=800.0 PL=0
MOVL C01015 V=800.0 PL=0
MOVL C01016 V=800.0 PL=0
MOVL C01017 V=800.0 PL=0
MOVL C01018 V=800.0 PL=0
MOVL C01019 V=800.0 PL=0
MOVL C01020 V=800.0 PL=0
MOVL C01021 V=800.0 PL=0
MOVL C01022 V=800.0 PL=0
MOVL C01023 V=800.0 PL=0
MOVL C01024 V=800.0 PL=0
MOVL C01025 V=800.0 PL=0
MOVL C01026 V=800.0 PL=0
MOVL C01027 V=800.0 PL=0
MOVL C01028 V=800.0 PL=0
MOVL C01029 V=800.0 PL=0
MOVL C01030 V=800.0 PL=0
MOVL C01031 V=800.0 PL=0
MOVL C01032 V=800.0 PL=0
MOVL C01033 V=800.0 PL=0
MOVL C01034 V=800.0 PL=0
MOVL C01035 V=800.0 PL=0
MOVL C01036 V=800.0 PL=0
MOVL C01037 V=800.0 PL=0
MOVL C01038 V=800.0 PL=0
MOVL C01039 V=800.0 PL=0
MOVL C01040 V=800.0 PL=0
MOVL C01041 V=800.0 PL=0
MOVL C01042 V=800.0 PL=0
MOVL C01043 V=800.0 PL=0
MOVL C01044 V=800.0 PL=0
MOVL C01045 V=800.0 PL=0
MOVL C01046 V=800.0 PL=0
MOVL C01047 V=800.0 PL=0
MOVL C01048 V=800.0 PL=0
MOVL C01049 V=800.0 PL=0
MOVL C01050 V=800.0 PL=0
MOVL C01051 V=800.0 PL=0
MOVL C01052 V=800.0 PL=0
MOVL C01053 V=800.0 PL=0
MOVL C01054 V=800.0 PL=0
MOVL C01055 V=800.0 PL=0
MOVL C01056 V=800.0 PL=0
MOVL C01057 V=800.0 PL=0
MOVL C01058 V=800.0 PL=0
MOVL C01059 V=800.0 PL=0
MOVL C01060 V=800.0 PL=0
MOVL C01061 V=800.0 PL=0
MOVL C01062 V=800.0 PL=0
MOVL C01063 V=800.0 PL=0
MOVL C01064 V=800.0 PL=0
MOVL C01065 V=800.0 PL=0
MOVL C01066 V=800.0 PL=0
MOVL C01067 V=800.0 PL=0
MOVL C01068 V=800.0 PL=0
MOVL C01069 V=800.0 PL=0
MOVL C01070 V=800.0 PL=0
MOVL C01071 V=800.0 PL=0
MOVL C01072 V=800.0 PL=0
MOVL C01073 V=800.0 PL=0
MOVL C01074 V=800.0 PL=0
MOVL C01075 V=800.0 PL=0
MOVL C01076 V=800.0 PL=0
MOVL C01077 V=800.0 PL=0
MOVL C01078 V=800.0 PL=0
MOVL C01079 V=800.0 PL=0
MOVL C01080 V=800.0 PL=0
MOVL C01081 V=800.0 PL=0
MOVL C01082 V=800.0 PL=0
MOVL C01083 V=800.0 PL=0
MOVL C01084 V=800.0 PL=0
MOVL C01085 V=800.0 PL=0
MOVL C01086 V=800.0 PL=0
MOVL C01087 V=800.0 PL=0
MOVL C01088 V=800.0 PL=0
MOVL C01089 V=800.0 PL=0
MOVL C01090 V=800.0 PL=0
MOVL C01091 V=800.0 PL=0
MOVL C01092 V=800.0 PL=0
MOVL C01093 V=800.0 PL=0
MOVL C01094 V=800.0 PL=0
MOVL C01095 V=800.0 PL=0
MOVL C01096 V=800.0 PL=0
MOVL C01097 V=800.0 PL=0
MOVL C01098 V=800.0 PL=0
MOVL C01099 V=800.0 PL=0
MOVL C01100 V=800.0 PL=0
MOVL C01101 V=800.0 PL=0
MOVL C01102 V=800.0 PL=0
MOVL C01103 V=800.0 PL=0
MOVL C01104 V=800.0 PL=0
MOVL C01105 V=800.0 PL=0
MOVL C01106 V=800.0 PL=0
MOVL C01107 V=800.0 PL=0
MOVL C01108 V=800.0 PL=0
MOVL C01109 V=800.0 PL=0
MOVL C01110 V=800.0 PL=0
MOVL C01111 V=800.0 PL=0
MOVL C01112 V=800.0 PL=0
MOVL C01113 V=800.0 PL=0
MOVL C01114 V=800.0 PL=0
MOVL C01115 V=800.0 PL=0
MOVL C01116 V=800.0 PL=0
MOVL C01117 V=800.0 PL=0
MOVL C01118 V=800.0 PL=0
MOVL C01119 V=800.0 PL=0
MOVL C01120 V=800.0 PL=0
MOVL C01121 V=800.0 PL=0
MOVL C01122 V=800.0 PL=0
MOVL C01123 V=800.0 PL=0
MOVL C01124 V=800.0 PL=0
MOVL C01125 V=800.0 PL=0
MOVL C01126 V=800.0 PL=0
MOVL C01127 V=800.0 PL=0
MOVL C01128 V=800.0 PL=0
MOVL C01129 V=800.0 PL=0
MOVL C01130 V=800.0 PL=0
MOVL C01131 V=800.0 PL=0
MOVL C01132 V=800.0 PL=0
MOVL C01133 V=800.0 PL=0
MOVL C01134 V=800.0 PL=0
MOVL C01135 V=800.0 PL=0
MOVL C01136 V=800.0 PL=0
MOVL C01137 V=800.0 PL=0
MOVL C01138 V=800.0 PL=0
MOVL C01139 V=800.0 PL=0
MOVL C01140 V=800.0 PL=0
MOVL C01141 V=800.0 PL=0
MOVL C01142 V=800.0 PL=0
MOVL C01143 V=800.0 PL=0
MOVL C01144 V=800.0 PL=0
MOVL C01145 V=800.0 PL=0
MOVL C01146 V=800.0 PL=0
MOVL C01147 V=800.0 PL=0
MOVL C01148 V=800.0 PL=0
MOVL C01149 V=800.0 PL=0
MOVL C01150 V=800.0 PL=0
MOVL C01151 V=800.0 PL=0
MOVL C01152 V=800.0 PL=0
MOVL C01153 V=800.0 PL=0
MOVL C01154 V=800.0 PL=0
MOVL C01155 V=800.0 PL=0
MOVL C01156 V=800.0 PL=0
MOVL C01157 V=800.0 PL=0
MOVL C01158 V=800.0 PL=0
MOVL C01159 V=800.0 PL=0
MOVL C01160 V=800.0 PL=0
MOVL C01161 V=800.0 PL=0
MOVL C01162 V=800.0 PL=0
MOVL C01163 V=800.0 PL=0
MOVL C01164 V=800.0 PL=0
MOVL C01165 V=800.0 PL=0
MOVL C01166 V=800.0 PL=0
MOVL C01167 V=800.0 PL=0
MOVL C01168 V=800.0 PL=0
MOVL C01169 V=800.0 PL=0
MOVL C01170 V=800.0 PL=0
MOVL C01171 V=800.0 PL=0
MOVL C01172 V=800.0 PL=0
MOVL C01173 V=800.0 PL=0
MOVL C01174 V=800.0 PL=0
MOVL C01175 V=800.0 PL=0
MOVL C01176 V=800.0 PL=0
MOVL C01177 V=800.0 PL=0
MOVL C01178 V=800.0 PL=0
MOVL C01179 V=800.0 PL=0
MOVL C01180 V=800.0 PL=0
MOVL C01181 V=800.0 PL=0
MOVL C01182 V=800.0 PL=0
MOVL C01183 V=800.0 PL=0
MOVL C01184 V=800.0 PL=0
MOVL C01185 V=800.0 PL=0
MOVL C01186 V=800.0 PL=0
MOVL C01187 V=800.0 PL=0
MOVL C01188 V=800.0 PL=0
MOVL C01189 V=800.0 PL=0
MOVL C01190 V=800.0 PL=0
MOVL C01191 V=800.0 PL=0
MOVL C01192 V=800.0 PL=0
MOVL C01193 V=800.0 PL=0
MOVL C01194 V=800.0 PL=0
MOVL C01195 V=800.0 PL=0
MOVL C01196 V=800.0 PL=0
MOVL C01197 V=800.0 PL=0
MOVL C01198 V=800.0 PL=0
MOVL C01199 V=800.0 PL=0
MOVL C01200 V=800.0 PL=0
MOVL C01201 V=800.0 PL=0
MOVL C01202 V=800.0 PL=0
MOVL C01203 V=800.0 PL=0
MOVL C01204 V=800.0 PL=0
MOVL C01205 V=800.0 PL=0
MOVL C01206 V=800.0 PL=0
MOVL C01207 V=800.0 PL=0
MOVL C01208 V=800.0 PL=0
MOVL C01209 V=800.0 PL=0
MOVL C01210 V=800.0 PL=0
MOVL C01211 V=800.0 PL=0
MOVL C01212 V=800.0 PL=0
MOVL C01213 V=800.0 PL=0
MOVL C01214 V=800.0 PL=0
MOVL C01215 V=800.0 PL=0
MOVL C01216 V=800.0 PL=0
MOVL C01217 V=800.0 PL=0
MOVL C01218 V=800.0 PL=0
MOVL C01219 V=800.0 PL=0
MOVL C01220 V=800.0 PL=0
MOVL C01221 V=800.0 PL=0
MOVL C01222 V=800.0 PL=0
MOVL C01223 V=800.0 PL=0
MOVL C01224 V=800.0 PL=0
MOVL C01225 V=800.0 PL=0
MOVL C01226 V=800.0 PL=0
MOVL C01227 V=800.0 PL=0
MOVL C01228 V=800.0 PL=0
MOVL C01229 V=800.0 PL=0
MOVL C01230 V=800.0 PL=0
MOVL C01231 V=800.0 PL=0
MOVL C01232 V=800.0 PL=0
MOVL C01233 V=800.0 PL=0
MOVL C01234 V=800.0 PL=0
MOVL C01235 V=800.0 PL=0
MOVL C01236 V=800.0 PL=0
MOVL C01237 V=800.0 PL=0
MOVL C01238 V=800.0 PL=0
MOVL C01239 V=800.0 PL=0
MOVL C01240 V=800.0 PL=0
MOVL C01241 V=800.0 PL=0
MOVL C01242 V=800.0 PL=0
MOVL C01243 V=800.0 PL=0
MOVL C01244 V=800.0 PL=0
MOVL C01245 V=800.0 PL=0
MOVL C01246 V=800.0 PL=0
MOVL C01247 V=800.0 PL=0
MOVL C01248 V=800.0 PL=0
MOVL C01249 V=800.0 PL=0
MOVL C01250 V=800.0 PL=0
MOVL C01251 V=800.0 PL=0
MOVL C01252 V=800.0 PL=0
MOVL C01253 V=800.0 PL=0
MOVL C01254 V=800.0 PL=0
MOVL C01255 V=800.0 PL=0
MOVL C01256 V=800.0 PL=0
MOVL C01257 V=800.0 PL=0
MOVL C01258 V=800.0 PL=0
MOVL C01259 V=800.0 PL=0
MOVL C01260 V=800.0 PL=0
MOVL C01261 V=800.0 PL=0
MOVL C01262 V=800.0 PL=0
MOVL C01263 V=800.0 PL=0
MOVL C01264 V=800.0 PL=0
MOVL C01265 V=800.0 PL=0
MOVL C01266 V=800.0 PL=0
MOVL C01267 V=800.0 PL=0
MOVL C01268 V=800.0 PL=0
MOVL C01269 V=800.0 PL=0
MOVL C01270 V=800.0 PL=0
MOVL C01271 V=800.0 PL=0
MOVL C01272 V=800.0 PL=0
MOVL C01273 V=800.0 PL=0
MOVL C01274 V=800.0 PL=0
MOVL C01275 V=800.0 PL=0
MOVL C01276 V=800.0 PL=0
MOVL C01277 V=800.0 PL=0
MOVL C01278 V=800.0 PL=0
MOVL C01279 V=800.0 PL=0
MOVL C01280 V=800.0 PL=0
MOVL C01281 V=800.0 PL=0
MOVL C01282 V=800.0 PL=0
MOVL C01283 V=800.0 PL=0
MOVL C01284 V=800.0 PL=0
MOVL C01285 V=800.0 PL=0
MOVL C01286 V=800.0 PL=0
MOVL C01287 V=800.0 PL=0
MOVL C01288 V=800.0 PL=0
MOVL C01289 V=800.0 PL=0
MOVL C01290 V=800.0 PL=0
MOVL C01291 V=800.0 PL=0
MOVL C01292 V=800.0 PL=0
MOVL C01293 V=800.0 PL=0
MOVL C01294 V=800.0 PL=0
MOVL C01295 V=800.0 PL=0
MOVL C01296 V=800.0 PL=0
MOVL C01297 V=800.0 PL=0
MOVL C01298 V=800.0 PL=0
MOVL C01299 V=800.0 PL=0
MOVL C01300 V=800.0 PL=0
MOVL C01301 V=800.0 PL=0
MOVL C01302 V=800.0 PL=0
MOVL C01303 V=800.0 PL=0
MOVL C01304 V=800.0 PL=0
MOVL C01305 V=800.0 PL=0
MOVL C01306 V=800.0 PL=0
MOVL C01307 V=800.0 PL=0
MOVL C01308 V=800.0 PL=0
MOVL C01309 V=800.0 PL=0
MOVL C01310 V=800.0 PL=0
MOVL C01311 V=800.0 PL=0
MOVL C01312 V=800.0 PL=0
MOVL C01313 V=800.0 PL=0
MOVL C01314 V=800.0 PL=0
MOVL C01315 V=800.0 PL=0
MOVL C01316 V=800.0 PL=0
MOVL C01317 V=800.0 PL=0
MOVL C01318 V=800.0 PL=0
MOVL C01319 V=800.0 PL=0
MOVL C01320 V=800.0 PL=0
MOVL C01321 V=800.0 PL=0
MOVL C01322 V=800.0 PL=0
MOVL C01323 V=800.0 PL=0
MOVL C01324 V=800.0 PL=0
MOVL C01325 V=800.0 PL=0
MOVL C01326 V=800.0 PL=0
MOVL C01327 V=800.0 PL=0
MOVL C01328 V=800.0 PL=0
MOVL C01329 V=800.0 PL=0
MOVL C01330 V=800.0 PL=0
MOVL C01331 V=800.0 PL=0
MOVL C01332 V=800.0 PL=0
MOVL C01333 V=800.0 PL=0
MOVL C01334 V=800.0 PL=0
MOVL C01335 V=800.0 PL=0
MOVL C01336 V=800.0 PL=0
MOVL C01337 V=800.0 PL=0
MOVL C01338 V=800.0 PL=0
MOVL C01339 V=800.0 PL=0
MOVL C01340 V=800.0 PL=0
MOVL C01341 V=800.0 PL=0
MOVL C01342 V=800.0 PL=0
MOVL C01343 V=800.0 PL=0
MOVL C01344 V=800.0 PL=0
MOVL C01345 V=800.0 PL=0
MOVL C01346 V=800.0 PL=0
MOVL C01347 V=800.0 PL=0
MOVL C01348 V=800.0 PL=0
MOVL C01349 V=800.0 PL=0
MOVL C01350 V=800.0 PL=0
MOVL C01351 V=800.0 PL=0
MOVL C01352 V=800.0 PL=0
MOVL C01353 V=800.0 PL=0
MOVL C01354 V=800.0 PL=0
MOVL C01355 V=800.0 PL=0
MOVL C01356 V=800.0 PL=0
MOVL C01357 V=800.0 PL=0
MOVL C01358 V=800.0 PL=0
MOVL C01359 V=800.0 PL=0
MOVL C01360 V=800.0 PL=0
MOVL C01361 V=800.0 PL=0
MOVL C01362 V=800.0 PL=0
MOVL C01363 V=800.0 PL=0
MOVL C01364 V=800.0 PL=0
MOVL C01365 V=800.0 PL=0
MOVL C01366 V=800.0 PL=0
MOVL C01367 V=800.0 PL=0
MOVL C01368 V=800.0 PL=0
MOVL C01369 V=800.0 PL=0
MOVL C01370 V=800.0 PL=0
MOVL C01371 V=800.0 PL=0
MOVL C01372 V=800.0 PL=0
MOVL C01373 V=800.0 PL=0
MOVL C01374 V=800.0 PL=0
MOVL C01375 V=800.0 PL=0
MOVL C01376 V=800.0 PL=0
MOVL C01377 V=800.0 PL=0
MOVL C01378 V=800.0 PL=0
MOVL C01379 V=800.0 PL=0
MOVL C01380 V=800.0 PL=0
MOVL C01381 V=800.0 PL=0
MOVL C01382 V=800.0 PL=0
MOVL C01383 V=800.0 PL=0
MOVL C01384 V=800.0 PL=0
MOVL C01385 V=800.0 PL=0
MOVL C01386 V=800.0 PL=0
MOVL C01387 V=800.0 PL=0
MOVL C01388 V=800.0 PL=0
MOVL C01389 V=800.0 PL=0
MOVL C01390 V=800.0 PL=0
MOVL C01391 V=800.0 PL=0
MOVL C01392 V=800.0 PL=0
MOVL C01393 V=800.0 PL=0
MOVL C01394 V=800.0 PL=0
MOVL C01395 V=800.0 PL=0
MOVL C01396 V=800.0 PL=0
MOVL C01397 V=800.0 PL=0
MOVL C01398 V=800.0 PL=0
MOVL C01399 V=800.0 PL=0
MOVL C01400 V=800.0 PL=0
MOVL C01401 V=800.0 PL=0
MOVL C01402 V=800.0 PL=0
MOVL C01403 V=800.0 PL=0
MOVL C01404 V=800.0 PL=0
MOVL C01405 V=800.0 PL=0
MOVL C01406 V=800.0 PL=0
MOVL C01407 V=800.0 PL=0
MOVL C01408 V=800.0 PL=0
MOVL C01409 V=800.0 PL=0
MOVL C01410 V=800.0 PL=0
MOVL C01411 V=800.0 PL=0
MOVL C01412 V=800.0 PL=0
MOVL C01413 V=800.0 PL=0
MOVL C01414 V=800.0 PL=0
MOVL C01415 V=800.0 PL=0
MOVL C01416 V=800.0 PL=0
MOVL C01417 V=800.0 PL=0
MOVL C01418 V=800.0 PL=0
MOVL C01419 V=800.0 PL=0
MOVL C01420 V=800.0 PL=0
MOVL C01421 V=800.0 PL=0
MOVL C01422 V=800.0 PL=0
MOVL C01423 V=800.0 PL=0
MOVL C01424 V=800.0 PL=0
MOVL C01425 V=800.0 PL=0
MOVL C01426 V=800.0 PL=0
MOVL C01427 V=800.0 PL=0
MOVL C01428 V=800.0 PL=0
MOVL C01429 V=800.0 PL=0
MOVL C01430 V=800.0 PL=0
MOVL C01431 V=800.0 PL=0
MOVL C01432 V=800.0 PL=0
MOVL C01433 V=800.0 PL=0
MOVL C01434 V=800.0 PL=0
MOVL C01435 V=800.0 PL=0
MOVL C01436 V=800.0 PL=0
MOVL C01437 V=800.0 PL=0
MOVL C01438 V=800.0 PL=0
MOVL C01439 V=800.0 PL=0
MOVL C01440 V=800.0 PL=0
MOVL C01441 V=800.0 PL=0
MOVL C01442 V=800.0 PL=0
MOVL C01443 V=800.0 PL=0
MOVL C01444 V=800.0 PL=0
MOVL C01445 V=800.0 PL=0
MOVL C01446 V=800.0 PL=0
MOVL C01447 V=800.0 PL=0
MOVL C01448 V=800.0 PL=0
MOVL C01449 V=800.0 PL=0
MOVL C01450 V=800.0 PL=0
MOVL C01451 V=800.0 PL=0
MOVL C01452 V=800.0 PL=0
MOVL C01453 V=800.0 PL=0
MOVL C01454 V=800.0 PL=0
MOVL C01455 V=800.0 PL=0
MOVL C01456 V=800.0 PL=0
MOVL C01457 V=800.0 PL=0
MOVL C01458 V=800.0 PL=0
MOVL C01459 V=800.0 PL=0
MOVL C01460 V=800.0 PL=0
MOVL C01461 V=800.0 PL=0
MOVL C01462 V=800.0 PL=0
MOVL C01463 V=800.0 PL=0
MOVL C01464 V=800.0 PL=0
MOVL C01465 V=800.0 PL=0
MOVL C01466 V=800.0 PL=0
MOVL C01467 V=800.0 PL=0
MOVL C01468 V=800.0 PL=0
MOVL C01469 V=800.0 PL=0
MOVL C01470 V=800.0 PL=0
MOVL C01471 V=800.0 PL=0
MOVL C01472 V=800.0 PL=0
MOVL C01473 V=800.0 PL=0
MOVL C01474 V=800.0 PL=0
MOVL C01475 V=800.0 PL=0
MOVL C01476 V=800.0 PL=0
MOVL C01477 V=800.0 PL=0
MOVL C01478 V=800.0 PL=0
MOVL C01479 V=800.0 PL=0
MOVL C01480 V=800.0 PL=0
MOVL C01481 V=800.0 PL=0
MOVL C01482 V=800.0 PL=0
MOVL C01483 V=800.0 PL=0
MOVL C01484 V=800.0 PL=0
MOVL C01485 V=800.0 PL=0
MOVL C01486 V=800.0 PL=0
MOVL C01487 V=800.0 PL=0
MOVL C01488 V=800.0 PL=0
MOVL C01489 V=800.0 PL=0
MOVL C01490 V=800.0 PL=0
MOVL C01491 V=800.0 PL=0
MOVL C01492 V=800.0 PL=0
MOVL C01493 V=800.0 PL=0
MOVL C01494 V=800.0 PL=0
MOVL C01495 V=800.0 PL=0
MOVL C01496 V=800.0 PL=0
MOVL C01497 V=800.0 PL=0
MOVL C01498 V=800.0 PL=0
MOVL C01499 V=800.0 PL=0
MOVL C01500 V=800.0 PL=0
MOVL C01501 V=800.0 PL=0
MOVL C01502 V=800.0 PL=0
MOVL C01503 V=800.0 PL=0
MOVL C01504 V=800.0 PL=0
MOVL C01505 V=800.0 PL=0
MOVL C01506 V=800.0 PL=0
MOVL C01507 V=800.0 PL=0
MOVL C01508 V=800.0 PL=0
MOVL C01509 V=800.0 PL=0
MOVL C01510 V=800.0 PL=0
MOVL C01511 V=800.0 PL=0
MOVL C01512 V=800.0 PL=0
MOVL C01513 V=800.0 PL=0
MOVL C01514 V=800.0 PL=0
MOVL C01515 V=800.0 PL=0
MOVL C01516 V=800.0 PL=0
MOVL C01517 V=800.0 PL=0
MOVL C01518 V=800.0 PL=0
MOVL C01519 V=800.0 PL=0
MOVL C01520 V=800.0 PL=0
MOVL C01521 V=800.0 PL=0
MOVL C01522 V=800.0 PL=0
MOVL C01523 V=800.0 PL=0
MOVL C01524 V=800.0 PL=0
MOVL C01525 V=800.0 PL=0
MOVL C01526 V=800.0 PL=0
MOVL C01527 V=800.0 PL=0
MOVL C01528 V=800.0 PL=0
MOVL C01529 V=800.0 PL=0
MOVL C01530 V=800.0 PL=0
MOVL C01531 V=800.0 PL=0
MOVL C01532 V=800.0 PL=0
MOVL C01533 V=800.0 PL=0
MOVL C01534 V=800.0 PL=0
MOVL C01535 V=800.0 PL=0
MOVL C01536 V=800.0 PL=0
MOVL C01537 V=800.0 PL=0
MOVL C01538 V=800.0 PL=0
MOVL C01539 V=800.0 PL=0
MOVL C01540 V=800.0 PL=0
MOVL C01541 V=800.0 PL=0
MOVL C01542 V=800.0 PL=0
MOVL C01543 V=800.0 PL=0
MOVL C01544 V=800.0 PL=0
MOVL C01545 V=800.0 PL=0
MOVL C01546 V=800.0 PL=0
MOVL C01547 V=800.0 PL=0
MOVL C01548 V=800.0 PL=0
MOVL C01549 V=800.0 PL=0
MOVL C01550 V=800.0 PL=0
MOVL C01551 V=800.0 PL=0
MOVL C01552 V=800.0 PL=0
MOVL C01553 V=800.0 PL=0
MOVL C01554 V=800.0 PL=0
MOVL C01555 V=800.0 PL=0
MOVL C01556 V=800.0 PL=0
MOVL C01557 V=800.0 PL=0
MOVL C01558 V=800.0 PL=0
MOVL C01559 V=800.0 PL=0
MOVL C01560 V=800.0 PL=0
MOVL C01561 V=800.0 PL=0
MOVL C01562 V=800.0 PL=0
MOVL C01563 V=800.0 PL=0
MOVL C01564 V=800.0 PL=0
MOVL C01565 V=800.0 PL=0
MOVL C01566 V=800.0 PL=0
MOVL C01567 V=800.0 PL=0
MOVL C01568 V=800.0 PL=0
MOVL C01569 V=800.0 PL=0
MOVL C01570 V=800.0 PL=0
MOVL C01571 V=800.0 PL=0
MOVL C01572 V=800.0 PL=0
MOVL C01573 V=800.0 PL=0
MOVL C01574 V=800.0 PL=0
MOVL C01575 V=800.0 PL=0
MOVL C01576 V=800.0 PL=0
MOVL C01577 V=800.0 PL=0
MOVL C01578 V=800.0 PL=0
MOVL C01579 V=800.0 PL=0
MOVL C01580 V=800.0 PL=0
MOVL C01581 V=800.0 PL=0
MOVL C01582 V=800.0 PL=0
MOVL C01583 V=800.0 PL=0
MOVL C01584 V=800.0 PL=0
MOVL C01585 V=800.0 PL=0
MOVL C01586 V=800.0 PL=0
MOVL C01587 V=800.0 PL=0
MOVL C01588 V=800.0 PL=0
MOVL C01589 V=800.0 PL=0
MOVL C01590 V=800.0 PL=0
MOVL C01591 V=800.0 PL=0
MOVL C01592 V=800.0 PL=0
MOVL C01593 V=800.0 PL=0
MOVL C01594 V=800.0 PL=0
MOVL C01595 V=800.0 PL=0
MOVL C01596 V=800.0 PL=0
MOVL C01597 V=800.0 PL=0
MOVL C01598 V=800.0 PL=0
MOVL C01599 V=800.0 PL=0
MOVL C01600 V=800.0 PL=0
MOVL C01601 V=800.0 PL=0
MOVL C01602 V=800.0 PL=0
MOVL C01603 V=800.0 PL=0
MOVL C01604 V=800.0 PL=0
MOVL C01605 V=800.0 PL=0
MOVL C01606 V=800.0 PL=0
MOVL C01607 V=800.0 PL=0
MOVL C01608 V=800.0 PL=0
MOVL C01609 V=800.0 PL=0
MOVL C01610 V=800.0 PL=0
MOVL C01611 V=800.0 PL=0
MOVL C01612 V=800.0 PL=0
MOVL C01613 V=800.0 PL=0
MOVL C01614 V=800.0 PL=0
MOVL C01615 V=800.0 PL=0
MOVL C01616 V=800.0 PL=0
MOVL C01617 V=800.0 PL=0
MOVL C01618 V=800.0 PL=0
MOVL C01619 V=800.0 PL=0
MOVL C01620 V=800.0 PL=0
MOVL C01621 V=800.0 PL=0
MOVL C01622 V=800.0 PL=0
MOVL C01623 V=800.0 PL=0
MOVL C01624 V=800.0 PL=0
MOVL C01625 V=800.0 PL=0
MOVL C01626 V=800.0 PL=0
MOVL C01627 V=800.0 PL=0
MOVL C01628 V=800.0 PL=0
MOVL C01629 V=800.0 PL=0
MOVL C01630 V=800.0 PL=0
MOVL C01631 V=800.0 PL=0
MOVL C01632 V=800.0 PL=0
MOVL C01633 V=800.0 PL=0
MOVL C01634 V=800.0 PL=0
MOVL C01635 V=800.0 PL=0
MOVL C01636 V=800.0 PL=0
MOVL C01637 V=800.0 PL=0
MOVL C01638 V=800.0 PL=0
MOVL C01639 V=800.0 PL=0
MOVL C01640 V=800.0 PL=0
MOVL C01641 V=800.0 PL=0
MOVL C01642 V=800.0 PL=0
MOVL C01643 V=800.0 PL=0
MOVL C01644 V=800.0 PL=0
MOVL C01645 V=800.0 PL=0
MOVL C01646 V=800.0 PL=0
MOVL C01647 V=800.0 PL=0
MOVL C01648 V=800.0 PL=0
MOVL C01649 V=800.0 PL=0
MOVL C01650 V=800.0 PL=0
MOVL C01651 V=800.0 PL=0
MOVL C01652 V=800.0 PL=0
MOVL C01653 V=800.0 PL=0
MOVL C01654 V=800.0 PL=0
MOVL C01655 V=800.0 PL=0
MOVL C01656 V=800.0 PL=0
MOVL C01657 V=800.0 PL=0
MOVL C01658 V=800.0 PL=0
MOVL C01659 V=800.0 PL=0
MOVL C01660 V=800.0 PL=0
MOVL C01661 V=800.0 PL=0
MOVL C01662 V=800.0 PL=0
MOVL C01663 V=800.0 PL=0
MOVL C01664 V=800.0 PL=0
MOVL C01665 V=800.0 PL=0
MOVL C01666 V=800.0 PL=0
MOVL C01667 V=800.0 PL=0
MOVL C01668 V=800.0 PL=0
MOVL C01669 V=800.0 PL=0
MOVL C01670 V=800.0 PL=0
MOVL C01671 V=800.0 PL=0
MOVL C01672 V=800.0 PL=0
MOVL C01673 V=800.0 PL=0
MOVL C01674 V=800.0 PL=0
MOVL C01675 V=800.0 PL=0
MOVL C01676 V=800.0 PL=0
MOVL C01677 V=800.0 PL=0
MOVL C01678 V=800.0 PL=0
MOVL C01679 V=800.0 PL=0
MOVL C01680 V=800.0 PL=0
MOVL C01681 V=800.0 PL=0
MOVL C01682 V=800.0 PL=0
MOVL C01683 V=800.0 PL=0
MOVL C01684 V=800.0 PL=0
MOVL C01685 V=800.0 PL=0
MOVL C01686 V=800.0 PL=0
MOVL C01687 V=800.0 PL=0
MOVL C01688 V=800.0 PL=0
MOVL C01689 V=800.0 PL=0
MOVL C01690 V=800.0 PL=0
MOVL C01691 V=800.0 PL=0
MOVL C01692 V=800.0 PL=0
MOVL C01693 V=800.0 PL=0
MOVL C01694 V=800.0 PL=0
MOVL C01695 V=800.0 PL=0
MOVL C01696 V=800.0 PL=0
MOVL C01697 V=800.0 PL=0
MOVL C01698 V=800.0 PL=0
MOVL C01699 V=800.0 PL=0
MOVL C01700 V=800.0 PL=0
MOVL C01701 V=800.0 PL=0
MOVL C01702 V=800.0 PL=0
MOVL C01703 V=800.0 PL=0
MOVL C01704 V=800.0 PL=0
MOVL C01705 V=800.0 PL=0
MOVL C01706 V=800.0 PL=0
MOVL C01707 V=800.0 PL=0
MOVL C01708 V=800.0 PL=0
MOVL C01709 V=800.0 PL=0
MOVL C01710 V=800.0 PL=0
MOVL C01711 V=800.0 PL=0
MOVL C01712 V=800.0 PL=0
MOVL C01713 V=800.0 PL=0
MOVL C01714 V=800.0 PL=0
MOVL C01715 V=800.0 PL=0
MOVL C01716 V=800.0 PL=0
MOVL C01717 V=800.0 PL=0
MOVL C01718 V=800.0 PL=0
MOVL C01719 V=800.0 PL=0
MOVL C01720 V=800.0 PL=0
MOVL C01721 V=800.0 PL=0
MOVL C01722 V=800.0 PL=0
MOVL C01723 V=800.0 PL=0
MOVL C01724 V=800.0 PL=0
MOVL C01725 V=800.0 PL=0
MOVL C01726 V=800.0 PL=0
MOVL C01727 V=800.0 PL=0
MOVL C01728 V=800.0 PL=0
MOVL C01729 V=800.0 PL=0
MOVL C01730 V=800.0 PL=0
MOVL C01731 V=800.0 PL=0
MOVL C01732 V=800.0 PL=0
MOVL C01733 V=800.0 PL=0
MOVL C01734 V=800.0 PL=0
MOVL C01735 V=800.0 PL=0
MOVL C01736 V=800.0 PL=0
MOVL C01737 V=800.0 PL=0
MOVL C01738 V=800.0 PL=0
MOVL C01739 V=800.0 PL=0
MOVL C01740 V=800.0 PL=0
MOVL C01741 V=800.0 PL=0
MOVL C01742 V=800.0 PL=0
MOVL C01743 V=800.0 PL=0
MOVL C01744 V=800.0 PL=0
MOVL C01745 V=800.0 PL=0
MOVL C01746 V=800.0 PL=0
MOVL C01747 V=800.0 PL=0
MOVL C01748 V=800.0 PL=0
MOVL C01749 V=800.0 PL=0
MOVL C01750 V=800.0 PL=0
MOVL C01751 V=800.0 PL=0
MOVL C01752 V=800.0 PL=0
MOVL C01753 V=800.0 PL=0
MOVL C01754 V=800.0 PL=0
MOVL C01755 V=800.0 PL=0
MOVL C01756 V=800.0 PL=0
MOVL C01757 V=800.0 PL=0
MOVL C01758 V=800.0 PL=0
MOVL C01759 V=800.0 PL=0
MOVL C01760 V=800.0 PL=0
MOVL C01761 V=800.0 PL=0
MOVL C01762 V=800.0 PL=0
MOVL C01763 V=800.0 PL=0
MOVL C01764 V=800.0 PL=0
MOVL C01765 V=800.0 PL=0
MOVL C01766 V=800.0 PL=0
MOVL C01767 V=800.0 PL=0
MOVL C01768 V=800.0 PL=0
MOVL C01769 V=800.0 PL=0
MOVL C01770 V=800.0 PL=0
MOVL C01771 V=800.0 PL=0
MOVL C01772 V=800.0 PL=0
MOVL C01773 V=800.0 PL=0
MOVL C01774 V=800.0 PL=0
MOVL C01775 V=800.0 PL=0
MOVL C01776 V=800.0 PL=0
MOVL C01777 V=800.0 PL=0
MOVL C01778 V=800.0 PL=0
MOVL C01779 V=800.0 PL=0
MOVL C01780 V=800.0 PL=0
MOVL C01781 V=800.0 PL=0
MOVL C01782 V=800.0 PL=0
MOVL C01783 V=800.0 PL=0
MOVL C01784 V=800.0 PL=0
MOVL C01785 V=800.0 PL=0
MOVL C01786 V=800.0 PL=0
MOVL C01787 V=800.0 PL=0
MOVL C01788 V=800.0 PL=0
MOVL C01789 V=800.0 PL=0
MOVL C01790 V=800.0 PL=0
MOVL C01791 V=800.0 PL=0
MOVL C01792 V=800.0 PL=0
MOVL C01793 V=800.0 PL=0
MOVL C01794 V=800.0 PL=0
MOVL C01795 V=800.0 PL=0
MOVL C01796 V=800.0 PL=0
MOVL C01797 V=800.0 PL=0
MOVL C01798 V=800.0 PL=0
MOVL C01799 V=800.0 PL=0
MOVL C01800 V=800.0 PL=0
MOVL C01801 V=800.0 PL=0
MOVL C01802 V=800.0 PL=0
MOVL C01803 V=800.0 PL=0
MOVL C01804 V=800.0 PL=0
MOVL C01805 V=800.0 PL=0
MOVL C01806 V=800.0 PL=0
MOVL C01807 V=800.0 PL=0
MOVL C01808 V=800.0 PL=0
MOVL C01809 V=800.0 PL=0
MOVL C01810 V=800.0 PL=0
MOVL C01811 V=800.0 PL=0
MOVL C01812 V=800.0 PL=0
MOVL C01813 V=800.0 PL=0
MOVL C01814 V=800.0 PL=0
MOVL C01815 V=800.0 PL=0
MOVL C01816 V=800.0 PL=0
MOVL C01817 V=800.0 PL=0
MOVL C01818 V=800.0 PL=0
MOVL C01819 V=800.0 PL=0
MOVL C01820 V=800.0 PL=0
MOVL C01821 V=800.0 PL=0
MOVL C01822 V=800.0 PL=0
MOVL C01823 V=800.0 PL=0
MOVL C01824 V=800.0 PL=0
MOVL C01825 V=800.0 PL=0
MOVL C01826 V=800.0 PL=0
MOVL C01827 V=800.0 PL=0
MOVL C01828 V=800.0 PL=0
MOVL C01829 V=800.0 PL=0
MOVL C01830 V=800.0 PL=0
MOVL C01831 V=800.0 PL=0
MOVL C01832 V=800.0 PL=0
MOVL C01833 V=800.0 PL=0
MOVL C01834 V=800.0 PL=0
MOVL C01835 V=800.0 PL=0
MOVL C01836 V=800.0 PL=0
MOVL C01837 V=800.0 PL=0
MOVL C01838 V=800.0 PL=0
MOVL C01839 V=800.0 PL=0
MOVL C01840 V=800.0 PL=0
MOVL C01841 V=800.0 PL=0
MOVL C01842 V=800.0 PL=0
MOVL C01843 V=800.0 PL=0
MOVL C01844 V=800.0 PL=0
MOVL C01845 V=800.0 PL=0
MOVL C01846 V=800.0 PL=0
MOVL C01847 V=800.0 PL=0
MOVL C01848 V=800.0 PL=0
MOVL C01849 V=800.0 PL=0
MOVL C01850 V=800.0 PL=0
MOVL C01851 V=800.0 PL=0
MOVL C01852 V=800.0 PL=0
MOVL C01853 V=800.0 PL=0
MOVL C01854 V=800.0 PL=0
MOVL C01855 V=800.0 PL=0
MOVL C01856 V=800.0 PL=0
MOVL C01857 V=800.0 PL=0
MOVL C01858 V=800.0 PL=0
MOVL C01859 V=800.0 PL=0
MOVL C01860 V=800.0 PL=0
MOVL C01861 V=800.0 PL=0
MOVL C01862 V=800.0 PL=0
MOVL C01863 V=800.0 PL=0
MOVL C01864 V=800.0 PL=0
MOVL C01865 V=800.0 PL=0
MOVL C01866 V=800.0 PL=0
MOVL C01867 V=800.0 PL=0
MOVL C01868 V=800.0 PL=0
MOVL C01869 V=800.0 PL=0
MOVL C01870 V=800.0 PL=0
MOVL C01871 V=800.0 PL=0
MOVL C01872 V=800.0 PL=0
MOVL C01873 V=800.0 PL=0
MOVL C01874 V=800.0 PL=0
MOVL C01875 V=800.0 PL=0
MOVL C01876 V=800.0 PL=0
MOVL C01877 V=800.0 PL=0
MOVL C01878 V=800.0 PL=0
MOVL C01879 V=800.0 PL=0
MOVL C01880 V=800.0 PL=0
MOVL C01881 V=800.0 PL=0
MOVL C01882 V=800.0 PL=0
MOVL C01883 V=800.0 PL=0
MOVL C01884 V=800.0 PL=0
MOVL C01885 V=800.0 PL=0
MOVL C01886 V=800.0 PL=0
MOVL C01887 V=800.0 PL=0
MOVL C01888 V=800.0 PL=0
MOVL C01889 V=800.0 PL=0
MOVL C01890 V=800.0 PL=0
MOVL C01891 V=800.0 PL=0
MOVL C01892 V=800.0 PL=0
MOVL C01893 V=800.0 PL=0
MOVL C01894 V=800.0 PL=0
MOVL C01895 V=800.0 PL=0
MOVL C01896 V=800.0 PL=0
MOVL C01897 V=800.0 PL=0
MOVL C01898 V=800.0 PL=0
MOVL C01899 V=800.0 PL=0
MOVL C01900 V=800.0 PL=0
MOVL C01901 V=800.0 PL=0
MOVL C01902 V=800.0 PL=0
MOVL C01903 V=800.0 PL=0
MOVL C01904 V=800.0 PL=0
MOVL C01905 V=800.0 PL=0
MOVL C01906 V=800.0 PL=0
MOVL C01907 V=800.0 PL=0
MOVL C01908 V=800.0 PL=0
MOVL C01909 V=800.0 PL=0
MOVL C01910 V=800.0 PL=0
MOVL C01911 V=800.0 PL=0
MOVL C01912 V=800.0 PL=0
MOVL C01913 V=800.0 PL=0
MOVL C01914 V=800.0 PL=0
MOVL C01915 V=800.0 PL=0
MOVL C01916 V=800.0 PL=0
MOVL C01917 V=800.0 PL=0
MOVL C01918 V=800.0 PL=0
MOVL C01919 V=800.0 PL=0
MOVL C01920 V=800.0 PL=0
MOVL C01921 V=800.0 PL=0
MOVL C01922 V=800.0 PL=0
MOVL C01923 V=800.0 PL=0
MOVL C01924 V=800.0 PL=0
MOVL C01925 V=800.0 PL=0
MOVL C01926 V=800.0 PL=0
MOVL C01927 V=800.0 PL=0
MOVL C01928 V=800.0 PL=0
MOVL C01929 V=800.0 PL=0
MOVL C01930 V=800.0 PL=0
MOVL C01931 V=800.0 PL=0
MOVL C01932 V=800.0 PL=0
MOVL C01933 V=800.0 PL=0
MOVL C01934 V=800.0 PL=0
MOVL C01935 V=800.0 PL=0
MOVL C01936 V=800.0 PL=0
MOVL C01937 V=800.0 PL=0
MOVL C01938 V=800.0 PL=0
MOVL C01939 V=800.0 PL=0
MOVL C01940 V=800.0 PL=0
MOVL C01941 V=800.0 PL=0
MOVL C01942 V=800.0 PL=0
MOVL C01943 V=800.0 PL=0
MOVL C01944 V=800.0 PL=0
MOVL C01945 V=800.0 PL=0
MOVL C01946 V=800.0 PL=0
MOVL C01947 V=800.0 PL=0
MOVL C01948 V=800.0 PL=0
MOVL C01949 V=800.0 PL=0
MOVL C01950 V=800.0 PL=0
MOVL C01951 V=800.0 PL=0
MOVL C01952 V=800.0 PL=0
MOVL C01953 V=800.0 PL=0
MOVL C01954 V=800.0 PL=0
MOVL C01955 V=800.0 PL=0
MOVL C01956 V=800.0 PL=0
MOVL C01957 V=800.0 PL=0
MOVL C01958 V=800.0 PL=0
MOVL C01959 V=800.0 PL=0
MOVL C01960 V=800.0 PL=0
MOVL C01961 V=800.0 PL=0
MOVL C01962 V=800.0 PL=0
MOVL C01963 V=800.0 PL=0
MOVL C01964 V=800.0 PL=0
MOVL C01965 V=800.0 PL=0
MOVL C01966 V=800.0 PL=0
MOVL C01967 V=800.0 PL=0
MOVL C01968 V=800.0 PL=0
MOVL C01969 V=800.0 PL=0
MOVL C01970 V=800.0 PL=0
MOVL C01971 V=800.0 PL=0
MOVL C01972 V=800.0 PL=0
MOVL C01973 V=800.0 PL=0
MOVL C01974 V=800.0 PL=0
MOVL C01975 V=800.0 PL=0
MOVL C01976 V=800.0 PL=0
MOVL C01977 V=800.0 PL=0
MOVL C01978 V=800.0 PL=0
MOVL C01979 V=800.0 PL=0
MOVL C01980 V=800.0 PL=0
MOVL C01981 V=800.0 PL=0
MOVL C01982 V=800.0 PL=0
MOVL C01983 V=800.0 PL=0
MOVL C01984 V=800.0 PL=0
MOVL C01985 V=800.0 PL=0
MOVL C01986 V=800.0 PL=0
MOVL C01987 V=800.0 PL=0
MOVL C01988 V=800.0 PL=0
MOVL C01989 V=800.0 PL=0
MOVL C01990 V=800.0 PL=0
MOVL C01991 V=800.0 PL=0
MOVL C01992 V=800.0 PL=0
MOVL C01993 V=800.0 PL=0
MOVL C01994 V=800.0 PL=0
MOVL C01995 V=800.0 PL=0
MOVL C01996 V=800.0 PL=0
MOVL C01997 V=800.0 PL=0
MOVL C01998 V=800.0 PL=0
MOVL C01999 V=800.0 PL=0
MOVL C02000 V=800.0 PL=0
MOVL C02001 V=800.0 PL=0
MOVL C02002 V=800.0 PL=0
MOVL C02003 V=800.0 PL=0
MOVL C02004 V=800.0 PL=0
MOVL C02005 V=800.0 PL=0
MOVL C02006 V=800.0 PL=0
MOVL C02007 V=800.0 PL=0
MOVL C02008 V=800.0 PL=0
MOVL C02009 V=800.0 PL=0
MOVL C02010 V=800.0 PL=0
MOVL C02011 V=800.0 PL=0
MOVL C02012 V=800.0 PL=0
MOVL C02013 V=800.0 PL=0
MOVL C02014 V=800.0 PL=0
MOVL C02015 V=800.0 PL=0
MOVL C02016 V=800.0 PL=0
MOVL C02017 V=800.0 PL=0
MOVL C02018 V=800.0 PL=0
MOVL C02019 V=800.0 PL=0
MOVL C02020 V=800.0 PL=0
MOVL C02021 V=800.0 PL=0
MOVL C02022 V=800.0 PL=0
MOVL C02023 V=800.0 PL=0
MOVL C02024 V=800.0 PL=0
MOVL C02025 V=800.0 PL=0
MOVL C02026 V=800.0 PL=0
MOVL C02027 V=800.0 PL=0
MOVL C02028 V=800.0 PL=0
MOVL C02029 V=800.0 PL=0
MOVL C02030 V=800.0 PL=0
MOVL C02031 V=800.0 PL=0
MOVL C02032 V=800.0 PL=0
MOVL C02033 V=800.0 PL=0
MOVL C02034 V=800.0 PL=0
MOVL C02035 V=800.0 PL=0
MOVL C02036 V=800.0 PL=0
MOVL C02037 V=800.0 PL=0
MOVL C02038 V=800.0 PL=0
MOVL C02039 V=800.0 PL=0
MOVL C02040 V=800.0 PL=0
MOVL C02041 V=800.0 PL=0
MOVL C02042 V=800.0 PL=0
MOVL C02043 V=800.0 PL=0
MOVL C02044 V=800.0 PL=0
MOVL C02045 V=800.0 PL=0
MOVL C02046 V=800.0 PL=0
MOVL C02047 V=800.0 PL=0
MOVL C02048 V=800.0 PL=0
MOVL C02049 V=800.0 PL=0
MOVL C02050 V=800.0 PL=0
MOVL C02051 V=800.0 PL=0
MOVL C02052 V=800.0 PL=0
MOVL C02053 V=800.0 PL=0
MOVL C02054 V=800.0 PL=0
MOVL C02055 V=800.0 PL=0
MOVL C02056 V=800.0 PL=0
MOVL C02057 V=800.0 PL=0
MOVL C02058 V=800.0 PL=0
MOVL C02059 V=800.0 PL=0
MOVL C02060 V=800.0 PL=0
MOVL C02061 V=800.0 PL=0
MOVL C02062 V=800.0 PL=0
MOVL C02063 V=800.0 PL=0
MOVL C02064 V=800.0 PL=0
MOVL C02065 V=800.0 PL=0
MOVL C02066 V=800.0 PL=0
MOVL C02067 V=800.0 PL=0
MOVL C02068 V=800.0 PL=0
MOVL C02069 V=800.0 PL=0
MOVL C02070 V=800.0 PL=0
MOVL C02071 V=800.0 PL=0
MOVL C02072 V=800.0 PL=0
MOVL C02073 V=800.0 PL=0
MOVL C02074 V=800.0 PL=0
MOVL C02075 V=800.0 PL=0
MOVL C02076 V=800.0 PL=0
MOVL C02077 V=800.0 PL=0
MOVL C02078 V=800.0 PL=0
MOVL C02079 V=800.0 PL=0
MOVL C02080 V=800.0 PL=0
MOVL C02081 V=800.0 PL=0
MOVL C02082 V=800.0 PL=0
MOVL C02083 V=800.0 PL=0
MOVL C02084 V=800.0 PL=0
MOVL C02085 V=800.0 PL=0
MOVL C02086 V=800.0 PL=0
MOVL C02087 V=800.0 PL=0
MOVL C02088 V=800.0 PL=0
MOVL C02089 V=800.0 PL=0
MOVL C02090 V=800.0 PL=0
MOVL C02091 V=800.0 PL=0
MOVL C02092 V=800.0 PL=0
MOVL C02093 V=800.0 PL=0
MOVL C02094 V=800.0 PL=0
MOVL C02095 V=800.0 PL=0
MOVL C02096 V=800.0 PL=0
MOVL C02097 V=800.0 PL=0
MOVL C02098 V=800.0 PL=0
MOVL C02099 V=800.0 PL=0
MOVL C02100 V=800.0 PL=0
MOVL C02101 V=800.0 PL=0
MOVL C02102 V=800.0 PL=0
MOVL C02103 V=800.0 PL=0
MOVL C02104 V=800.0 PL=0
MOVL C02105 V=800.0 PL=0
MOVL C02106 V=800.0 PL=0
MOVL C02107 V=800.0 PL=0
MOVL C02108 V=800.0 PL=0
MOVL C02109 V=800.0 PL=0
MOVL C02110 V=800.0 PL=0
MOVL C02111 V=800.0 PL=0
MOVL C02112 V=800.0 PL=0
MOVL C02113 V=800.0 PL=0
MOVL C02114 V=800.0 PL=0
MOVL C02115 V=800.0 PL=0
